(* CODESYS project EngineeringToolbox.library
   Company: Beckhoff Electronics Mfg
   DefaultNamespace: ET
   Version: 3.1.0.13
   Placeholder: ET
   Author: Daniel Schlingmann
   Description: Engineering Toolbox Library
      
      The library is provided "as-is" for TwinCAT3.1 by the Beckhoff Industry Management for Electronics Manufacturing.
      Please check the function "DisclaimerStatement : WSTRING[1500]"
   Title: EngineeringToolbox

Project tree, tasks and I/O mapping:
  libraries: Tc2_BackupRestoreEL6900, * (Beckhoff Automation GmbH); Tc2_Drive, * (Beckhoff Automation GmbH); Tc2_EtherCAT, * (Beckhoff Automation GmbH); Tc2_IoFunctions, * (Beckhoff Automation GmbH); Tc2_Math, * (Beckhoff Automation GmbH); Tc2_MC2, * (Beckhoff Automation GmbH); Tc2_MC2_Camming, * (Beckhoff Automation GmbH); Tc2_MC2_Drive, * (Beckhoff Automation GmbH); Tc2_MC2_FlyingSaw, * (Beckhoff Automation GmbH); Tc2_MDP, * (Beckhoff Automation GmbH); Tc2_ModbusRTU, * (Beckhoff Automation GmbH); Tc2_ModbusSrv, * (Beckhoff Automation GmbH); Tc2_NC, * (Beckhoff Automation GmbH); Tc2_NCI, * (Beckhoff Automation GmbH); Tc2_NcKinematicTransformation, * (Beckhoff Automation GmbH); Tc2_PlcInterpolation, * (Beckhoff Automation GmbH); Tc2_SerialCom, * (Beckhoff Automation GmbH); Tc2_Smtp, * (Beckhoff Automation GmbH); Tc2_Standard, * (Beckhoff Automation GmbH); Tc2_SUPS, * (Beckhoff Automation GmbH); Tc2_System, * (Beckhoff Automation GmbH); Tc2_TcpIp, * (Beckhoff Automation GmbH); Tc2_Utilities, * (Beckhoff Automation GmbH); Tc2_XmlDataSrv, * (Beckhoff Automation GmbH); Tc3_Module, * (Beckhoff Automation GmbH)
  GVLs/
    global variables Gvl
    global variables PARAM
  POUs/
    _Miscellaneous/
      64BitFunctions/
        function CLEARBIT64 [ST]
        function CSETBIT64 [ST]
        function GETBIT64 [ST]
        function SETBIT64 [ST]
      Conversions/
        function ADSERROR_TO_HRESULT [ST]
        function ADSERROR_TO_WIN32ERROR [ST]
        function ADSERROR_TO_WSERROR [ST]
        function C_TO_F [ST]
        function DEGREES_TO_RPM [ST]
        function DWORD_TO_REAL_EX [ST]
        function F_TO_C [ST]
        function GF_TO_N [ST]
        function HRESULT_TO_ADSERROR [ST]
        function LWORD_TO_LREAL_EX [ST]
        function MMIN_TO_MMS [ST]
        function MMS_TO_MMIN [ST]
        function N_TO_GF [ST]
        function REAL_TO_FMLREAL [ST]
        function RPM_TO_DEGREES [ST]
        function SWAP_BYTES_OF_WORDS [ST]
        function SWAP_WORDS_OF_DWORD [ST]
        function SWAP_WORDS_OF_LWORD [ST]
        function TO_FMLREAL [ST]
      function CAM [ST]
      function CAM3D [ST]
      data type COLOR
      data type eLCID
      function block ERROR_HDL [ST]: reset
      function block FbBase [ST]
      function block FbBaseExt [ST]
      function block FbBaseOutputs [ST]
      function getNoOfBits [ST]
      data type LCID
      function LOGx [ST]
      function nextIdx [ST]
      function block OEECalculation [ST]: addBadUnits, addGoodUnits, reset
      function polynomial [ST]
      function block RF_TRIG [ST]
      function scale [ST]
      function block SEQUENCE_HDL [ST]: abort, active, finish, incState, reset, resetWithErrHdl, set, ton_BT, ton_PT, tonOFF, tonON, tonRUN
      function setNoOfBits [ST]
      data type TC_VN_COLORS
      function block TEST_FB [ST]
      function block TOGGLE [ST]: CLK, RESET, SET
      data type U_32BIT_DATATYPE
      data type U_64BIT_DATATYPE
      function WIN [ST]
    BoundsCheck/
      function boundsError [ST]
      function boundsOK [ST]
      function block CheckBoundsInfo [ST]: reset, setErrorLower, setErrorUpper
    Connectivity/
      ADS/
        function block AdsDataExchange [ST]
      TF625x-Modbus/
        Master/
          _Components/
            function block ModbusJob [ST]: init
            function block ModbusSlaveCom [ST]: deleteData
          TF6250-ModbusTcpServer/
            TCP/
              function block ModbusTcpMaster [ST]: getNextJob, getNextSlave, reset, startJob
            UDP/
              function block ModbusUdpMaster [ST]: getNextJob, getNextSlave, reset, startJob
          TF6255-ModbusRtu/
            function block ModbusRtuMaster22B [ST]: getNextJob, getNextSlave, reset, startJob
            function block ModbusRtuMaster5B [ST]: getNextJob, getNextSlave, reset, startJob
            function block ModbusRtuMasterPC [ST]: getNextJob, getNextSlave, reset, startJob
        Slave/
          function block ModbusSlaveBase [ST]: evaluation, initJobs, prepareWriteData, run
      TF6310-TcpServer/
        TCP/
          function block TCPSendRecCtrl [ST]: optDoNotRestartReceiveCyclic, receive, send
          function block TCPServerCtrl [ST]
          function block TCPSocketCtrl [ST]: accept, close, closeAll, connect, listen
        UDP/
          function block UDPSendRecCtrl [ST]: optDoNotRestartReceiveCylic, receive, send
          function block UDPServerCtrl [ST]
          function block UDPSocketCtrl [ST]: close, closeAll, create
      TF6340-SerialCom/
        function block ComPortBackground [ST]: reset
        function block ComPortSendRec [ST]: clearBuffer, optClearBuffer, optEnableStringMode, optRemovePrefix, optRemoveSuffix, receiveData, receiveStr, reset, sendData, sendStr
      function isValidIPv4Addr [ST]
      data type U_IPv4Addr
    ControllerTools/
      function block AverageFilter [ST]: clear, insert
      function block PIDController [ST]: reset, synchronize
      function block PT1Filter [ST]: reset, synchronize
      function signum [ST]
      function block SlewRateLimitter [ST]: synchronize
      function block SlidingAverage [ST]: reset
      function block SlidingAverageExt [ST]: FB_exit, reset
      function block ThreePointController [ST]: reset, synchronize
    DataBuffer/
      Fifo/
        function block Fifo [ST]: clear, clearByDataSet, dequeue, enqueue, isEnqueued, isNextEntry, readEntry, reset
        function block FifoBase [ST]: _clear, _clearByDataSet, _dequeue, _enqueue, _isEnqueued, _isNextEntry, _readEntry, _reset
        function block FifoExt [ST]: allocate, clear, clearByDataSet, dequeue, enqueue, FB_exit, isEnqueued, isNextEntry, readEntry, reset
        function block FifoLRealSimple [ST]: clear, clearByDataSet, dequeue, enqueue, isEnqueued, isNextEntry, readEntry, reset
      Ringbuffer/
        function block Ringbuffer [ST]: dequeue, dequeueStream, enqueue, enqueueStream, reset
        function block RingbufferBase [ST]: _dequeue, _dequeueStream, _enqueue, _enqueueStream, _reset
        function block RingbufferByteSimple [ST]: dequeue, dequeueStream, enqueue, enqueueStream, reset
        function block RingbufferCharSimple [ST]: dequeue, dequeueStream, enqueue, enqueueStream, reset
        function block RingbufferExt [ST]: allocate, dequeue, dequeueStream, enqueue, enqueueStream, FB_exit, reset
        function block RingbufferLRealSimple [ST]: dequeue, dequeueStream, enqueue, enqueueStream, reset
      function block DataFileLogger [ST]: addData, addString, optKeepFileOnError, optStartNewFile
      function block DoubleBuffer [ST]: addData, addString, allocate, copyData, FB_exit, fillLevel, reset, setReadyToRead, swapBuffer
      function block Quicksort [ST]: allocate, byDINT, byDINT_Bubble, byINT, byLREAL, byLTIME, byREAL, bySTRING, byTIME, byUINT, byUSINT, byWSTRING, FB_exit
    EventLogger/
      ReadEvents/
        data type EVENTLOG_READ_DATA
        data type EVENTLOG_READ_HANDLEINFO
        data type EVENTLOG_READ_STREAM
        data type EVENTLOG_READ_STREAM_DATA_RAW
        data type EVENTLOG_READ_STREAM_DATA_RAW_EX
        function block EventlogRead [ST]: optGetHostNameForEachEvent, optUseStateForTimestamp
      TriggerEvents/
        function block EventHandling [ST]
        function EventHandlingConfirmIsReq [ST]
        function block EventHandlingGrp10 [ST]: confirm, confirmIsReq, isActive
        function block EventHandlingGrp25 [ST]: confirm, confirmIsReq, isActive
        function block EventHandlingGrp50 [ST]: confirm, confirmIsReq, isActive
        function block EventHandlingGrpCustomized [ST]: confirm
        function block EventHandlingStatisticInfo [ST]: classAlarmActive, classHintActive, classInstructionActive, classMaintenanceActive, classMessageActive, classNoneActive, classParamErrorActive, classStateinfoActive, classWarningActive, clear, countIn, countOut, initEvent, isClassActive, isConfirmReqActive, isPriorityActive
      data type EVENT_HANDLING_CONFIG
      function block EventsWriteToLogbook [ST]: _formatMsg
      function getEventClassPriority [ST]
      function getEventClassText [ST]
      data type SOURCE_ID
    Fieldbus/
      CANopen/
        function block CANopenMasterDiag [ST]
        function block CANopenMasterIO [ST]: setName
      EtherCAT/
        _Components/
          data type EC_MASTER_DEVICE_STATE
          data type EC_SLAVE_DIAG_INFO_DATA
          function block EcMasterIO [ST]
          function block EcMasterSupervisor [ST]: optClearCRCErrorCounter, optClearLostFramesCounter, optClearTCRXErrCounter, optForceDevReset
          function block EcSlavesDiag [ST]: allocate, FB_exit, optReadScannedSlaves, optSortInfoData, optUpdateConfigData, optUpdateTopoData, sortList
          function block EcSlaveSupervisor [ST]
        function block EcCoEReadNewestDiagMsg [ST]: msgSevyIsError, msgSevyIsInfo, msgSevyIsWarning
        function block EcDiagBase [ST]
        function block EcDiagBase_wEvents [ST]: _callEvents, confirm
      Profibus/
        function block ProfibusMasterDiag [ST]
        function block ProfibusMasterIO [ST]
      Profinet/
        function block ProfinetControllerIO [ST]
        function block ProfinetControllerIO_wEvents [ST]
        function block ProfinetDeviceIO [ST]
    FileHandling/
      Basic/
        function block FileHandling [ST]: close, createDir, delete, gets, isEoF, open, puts, read, removeDir, rename, seek, tell, write
        function block ReadDirSimple [ST]
        function block ReadDirSimpleExt [ST]
      TF6421-XmlServer/
        function block XmlReadWrite [ST]: read, write
        function block XmlReadWriteWithBackupFile [ST]: FB_exit, optEnableAutoSave, optEnableBackupFile, read, write
    IO/
      _EcSlaveFWUpdater/
        function block EcSlaveDevFWUpdater [ST]
      _EcSlaveInfoDataIO/
        function block EcSlaveInfoData [ST]: rInfoData
        function block EcSlaveInfoDataExt [ST]
        interface I_EcSlaveInfoData: rInfoData
      _ItfActuators/
        interface I_ActuatorBase: inError, isBusy, isOff, noFeed, ok, reset, switchOff
        interface I_ActuatorEnableDisable: isDisabled, isEnabled, setDisable, setEnable
        interface I_ActuatorFwdBwd: backwardStarted, forwardStarted, startBackward, startForward
        interface I_ActuatorFwdRev: forwardStarted, reverseStarted, startForward, startReverse
        interface I_ActuatorLeftRight: leftOk, rightOk, toTheLeft, toTheRight
        interface I_ActuatorOnOff: isOn, switchOn
        interface I_ActuatorOpenClose: isClosed, isOpened, setClose, setOpen
        interface I_ActuatorPosNeg: negativeOk, negativeOn, positiveOk, positiveOn
        interface I_ActuatorStartStop: isStarted, isStopped, start, stop
        interface I_ActuatorUpDown: downOk, moveDown, moveUp, upOK
        interface I_ActuatorWorkBase: isInBasePos, isInWorkPos, moveToBasePos, moveToWorkPos
      Cylinder/
        function block Cylinder [ST]: _readSensors, _runtimeChk, _writeStatus, enable, moveToBasePos, moveToWorkPos, reset, switchOff, optDisableLogicError, optDisableSensorBasepos, optDisableSensorWorkpos, optEnableImpulsValveFnc, optInvertSensorBasepos, optInvertSensorWorkpos, optSwapSensorStatus, inError, isBusy, isInBasePos, isInWorkPos, isOff, noFeed, ok, rCylinder, simulation
        function block CylinderExt [ST]: _runtimeChk
        function block CylinderType4 [ST]: _readSensors
        interface I_Cylinder: enable, rCylinder, simulation
      Drives/
        CoE/
          EL72xx/
            function block AxDriveCoE [ST]
            function block AxDriveCoE_EL72xxParam [ST]: deviceAddrIsValid, getValue, seqRead, seqWrite, setValue
            function block AxDriveCoE_wEvents [ST]: _callEvents, confirm, optDisabledRemoteCntrNotActive, optDisableIntLimitWarning
            function block CiA_DS402StatuswordEx7xxx [ST]: readStatusword
          function block CiA_DS402Controlword [ST]: createControlword
          function block CiA_DS402Statusword [ST]: readStatusword
          data type eCiA_DS402_CONTROL_CMD
          data type eCiA_DS402_STATUS_STATE
        DC/
          Ey73xx/
            function block AxDriveDC [ST]
            function block AxDriveDC_wEvents [ST]: _callEvents, confirm
        SoE/
          Ax5000ParamSTRUCTs/
            P/
              data type AX5000_P_0001
              data type AX5000_P_0002
              data type AX5000_P_0003
              data type AX5000_P_0004
              data type AX5000_P_0009
              data type AX5000_P_0010
              data type AX5000_P_0020
              data type AX5000_P_0021
              data type AX5000_P_0040
              data type AX5000_P_0050
              data type AX5000_P_0051
              data type AX5000_P_0052
              data type AX5000_P_0053
              data type AX5000_P_0054
              data type AX5000_P_0055
              data type AX5000_P_0056
              data type AX5000_P_0057
              data type AX5000_P_0058
              data type AX5000_P_0059
              data type AX5000_P_0060
              data type AX5000_P_0061
              data type AX5000_P_0062
              data type AX5000_P_0063
              data type AX5000_P_0064
              data type AX5000_P_0065
              data type AX5000_P_0066
              data type AX5000_P_0067
              data type AX5000_P_0068
              data type AX5000_P_0069
              data type AX5000_P_0070
              data type AX5000_P_0071
              data type AX5000_P_0072
              data type AX5000_P_0073
              data type AX5000_P_0074
              data type AX5000_P_0075
              data type AX5000_P_0076
              data type AX5000_P_0077
              data type AX5000_P_0078
              data type AX5000_P_0088
              data type AX5000_P_0089
              data type AX5000_P_0090
              data type AX5000_P_0091
              data type AX5000_P_0092
              data type AX5000_P_0093
              data type AX5000_P_0096
              data type AX5000_P_0097
              data type AX5000_P_0098_beckhoff
              data type AX5000_P_0098_beckhoff_electrical_data
              data type AX5000_P_0099
              data type AX5000_P_0100
              data type AX5000_P_0101
              data type AX5000_P_0102
              data type AX5000_P_0103
              data type AX5000_P_0104
              data type AX5000_P_0105
              data type AX5000_P_0106
              data type AX5000_P_0107
              data type AX5000_P_0108
              data type AX5000_P_0109
              data type AX5000_P_0110
              data type AX5000_P_0111
              data type AX5000_P_0112
              data type AX5000_P_0113
              data type AX5000_P_0114
              data type AX5000_P_0115
              data type AX5000_P_0116
              data type AX5000_P_0117
              data type AX5000_P_0118
              data type AX5000_P_0119
              data type AX5000_P_0125
              data type AX5000_P_0126
              data type AX5000_P_0127
              data type AX5000_P_0128
              data type AX5000_P_0150
              data type AX5000_P_0151
              data type AX5000_P_0152
              data type AX5000_P_0153
              data type AX5000_P_0154
              data type AX5000_P_0155
              data type AX5000_P_0158
              data type AX5000_P_0159
              data type AX5000_P_0160
              data type AX5000_P_0161
              data type AX5000_P_0162
              data type AX5000_P_0163
              data type AX5000_P_0165
              data type AX5000_P_0166
              data type AX5000_P_0167
              data type AX5000_P_0168
              data type AX5000_P_0169
              data type AX5000_P_0170
              data type AX5000_P_0171
              data type AX5000_P_0180
              data type AX5000_P_0181
              data type AX5000_P_0182
              data type AX5000_P_0183
              data type AX5000_P_0184
              data type AX5000_P_0185
              data type AX5000_P_0188
              data type AX5000_P_0189
              data type AX5000_P_0192
              data type AX5000_P_0193
              data type AX5000_P_0196
              data type AX5000_P_0198
              data type AX5000_P_0199
              data type AX5000_P_0200
              data type AX5000_P_0201
              data type AX5000_P_0202
              data type AX5000_P_0203
              data type AX5000_P_0204
              data type AX5000_P_0205
              data type AX5000_P_0206
              data type AX5000_P_0207
              data type AX5000_P_0208
              data type AX5000_P_0209
              data type AX5000_P_0210
              data type AX5000_P_0211
              data type AX5000_P_0212
              data type AX5000_P_0213
              data type AX5000_P_0214
              data type AX5000_P_0215
              data type AX5000_P_0216
              data type AX5000_P_0217
              data type AX5000_P_0218
              data type AX5000_P_0219
              data type AX5000_P_0220
              data type AX5000_P_0221
              data type AX5000_P_0250
              data type AX5000_P_0251
              data type AX5000_P_0252
              data type AX5000_P_0253
              data type AX5000_P_0254
              data type AX5000_P_0255
              data type AX5000_P_0256
              data type AX5000_P_0270
              data type AX5000_P_0271
              data type AX5000_P_0272
              data type AX5000_P_0273
              data type AX5000_P_0274
              data type AX5000_P_0275
              data type AX5000_P_0276
              data type AX5000_P_0277
              data type AX5000_P_0278
              data type AX5000_P_0300
              data type AX5000_P_0301
              data type AX5000_P_0302
              data type AX5000_P_0303
              data type AX5000_P_0304
              data type AX5000_P_0305
              data type AX5000_P_0306
              data type AX5000_P_0307
              data type AX5000_P_0308
              data type AX5000_P_0309
              data type AX5000_P_0310
              data type AX5000_P_0311
              data type AX5000_P_0312
              data type AX5000_P_0313
              data type AX5000_P_0314
              data type AX5000_P_0315
              data type AX5000_P_0316
              data type AX5000_P_0317
              data type AX5000_P_0320
              data type AX5000_P_0321
              data type AX5000_P_0322
              data type AX5000_P_0323
              data type AX5000_P_0324
              data type AX5000_P_0325
              data type AX5000_P_0326
              data type AX5000_P_0350
              data type AX5000_P_0351
              data type AX5000_P_0352
              data type AX5000_P_0353
              data type AX5000_P_0354
              data type AX5000_P_0356
              data type AX5000_P_0360
              data type AX5000_P_0361
              data type AX5000_P_0400
              data type AX5000_P_0401
              data type AX5000_P_0402
              data type AX5000_P_0451
              data type AX5000_P_0452
              data type AX5000_P_0453
              data type AX5000_P_0454
              data type AX5000_P_0455
              data type AX5000_P_0456
              data type AX5000_P_0457
              data type AX5000_P_0458
              data type AX5000_P_0459
              data type AX5000_P_0460
              data type AX5000_P_0461
              data type AX5000_P_0462
              data type AX5000_P_0463
              data type AX5000_P_0464
              data type AX5000_P_0502
              data type AX5000_P_0503
              data type AX5000_P_0504
              data type AX5000_P_0505
              data type AX5000_P_0511
              data type AX5000_P_0512
              data type AX5000_P_0513
              data type AX5000_P_0514
              data type AX5000_P_0515
              data type AX5000_P_0516
              data type AX5000_P_0517
              data type AX5000_P_0518
              data type AX5000_P_0552
              data type AX5000_P_0553
              data type AX5000_P_0554
              data type AX5000_P_0555
              data type AX5000_P_0556
              data type AX5000_P_0557
              data type AX5000_P_0558
              data type AX5000_P_0601
              data type AX5000_P_0602
              data type AX5000_P_0610
              data type AX5000_P_0611
              data type AX5000_P_0800
              data type AX5000_P_0801
              data type AX5000_P_0802
              data type AX5000_P_0804
              data type AX5000_P_0805
              data type AX5000_P_0806
              data type AX5000_P_0810
              data type AX5000_P_0811
              data type AX5000_P_0850
              data type AX5000_P_0851
              data type AX5000_P_0900
              data type AX5000_P_0901
              data type AX5000_P_0902
              data type AX5000_P_0904
              data type AX5000_P_0905
              data type AX5000_P_0906
              data type AX5000_P_0912
              data type AX5000_P_1000
              data type AX5000_P_1001
              data type AX5000_P_1002
              data type AX5000_P_1003
              data type AX5000_P_1004
              data type AX5000_P_1005
              data type AX5000_P_1006
              data type AX5000_P_1007
              data type AX5000_P_1008
              data type AX5000_P_1009
              data type AX5000_P_1010
              data type AX5000_P_1011
              data type AX5000_P_1012
              data type AX5000_P_1020
              data type AX5000_P_1021
              data type AX5000_P_1022
              data type AX5000_P_2000
              data type AX5000_P_2001
              data type AX5000_P_2002
            S/
              data type AX5000_S_0001
              data type AX5000_S_0002
              data type AX5000_S_0007
              data type AX5000_S_0011
              data type AX5000_S_0012
              data type AX5000_S_0013
              data type AX5000_S_0015
              data type AX5000_S_0016
              data type AX5000_S_0017
              data type AX5000_S_0018
              data type AX5000_S_0024
              data type AX5000_S_0029
              data type AX5000_S_0030
              data type AX5000_S_0031
              data type AX5000_S_0032
              data type AX5000_S_0033
              data type AX5000_S_0034
              data type AX5000_S_0035
              data type AX5000_S_0036
              data type AX5000_S_0037
              data type AX5000_S_0040
              data type AX5000_S_0043
              data type AX5000_S_0044
              data type AX5000_S_0045
              data type AX5000_S_0046
              data type AX5000_S_0047
              data type AX5000_S_0048
              data type AX5000_S_0051
              data type AX5000_S_0053
              data type AX5000_S_0055
              data type AX5000_S_0076
              data type AX5000_S_0079
              data type AX5000_S_0080
              data type AX5000_S_0081
              data type AX5000_S_0082
              data type AX5000_S_0083
              data type AX5000_S_0084
              data type AX5000_S_0085
              data type AX5000_S_0086
              data type AX5000_S_0091
              data type AX5000_S_0092
              data type AX5000_S_0095
              data type AX5000_S_0099
              data type AX5000_S_0100
              data type AX5000_S_0101
              data type AX5000_S_0103
              data type AX5000_S_0104
              data type AX5000_S_0106
              data type AX5000_S_0107
              data type AX5000_S_0109
              data type AX5000_S_0110
              data type AX5000_S_0111
              data type AX5000_S_0112
              data type AX5000_S_0113
              data type AX5000_S_0119
              data type AX5000_S_0120
              data type AX5000_S_0124
              data type AX5000_S_0126
              data type AX5000_S_0130
              data type AX5000_S_0131
              data type AX5000_S_0134
              data type AX5000_S_0135
              data type AX5000_S_0136
              data type AX5000_S_0137
              data type AX5000_S_0143
              data type AX5000_S_0149
              data type AX5000_S_0159
              data type AX5000_S_0160
              data type AX5000_S_0161
              data type AX5000_S_0162
              data type AX5000_S_0163
              data type AX5000_S_0169
              data type AX5000_S_0170
              data type AX5000_S_0179
              data type AX5000_S_0185
              data type AX5000_S_0186
              data type AX5000_S_0187
              data type AX5000_S_0188
              data type AX5000_S_0189
              data type AX5000_S_0196
              data type AX5000_S_0200
              data type AX5000_S_0201
              data type AX5000_S_0203
              data type AX5000_S_0204
              data type AX5000_S_0206
              data type AX5000_S_0207
              data type AX5000_S_0216
              data type AX5000_S_0217
              data type AX5000_S_0219
              data type AX5000_S_0254
              data type AX5000_S_0256
              data type AX5000_S_0257
              data type AX5000_S_0267
              data type AX5000_S_0273
              data type AX5000_S_0274
              data type AX5000_S_0292
              data type AX5000_S_0295
              data type AX5000_S_0296
              data type AX5000_S_0347
              data type AX5000_S_0348
              data type AX5000_S_0372
              data type AX5000_S_0374
              data type AX5000_S_0375
              data type AX5000_S_0380
              data type AX5000_S_0381
              data type AX5000_S_0383
              data type AX5000_S_0384
              data type AX5000_S_0390
              data type AX5000_S_0403
              data type AX5000_S_0405
              data type AX5000_S_0409
              data type AX5000_S_0410
              data type AX5000_S_0429
              data type AX5000_S_0432
              data type AX5000_S_0435
              data type AX5000_S_0436
          function block Ax580x [ST]
          function block AxDriveSoE_Ax5000 [ST]: break, refreshStatus, reset
          function block AxDriveSoE_Ax5000CalcPower [ST]: get_P_WORD, get_S_WORD
          function block AxDriveSoE_Ax5000CommutationCalib [ST]: optP98IsEmpty, optReadOnly
          function block AxDriveSoE_Ax5000Param [ST]: deviceAddrIsValid, getValue, seqRead, seqWrite, setValue
          function block AxDriveSoE_Ax5000SwitchParamSet [ST]: setNewParam
          function block AxDriveSoE_Ax5000wEvents [ST]: _callEvents, confirm
          function block AxDriveSoE_Rexroth [ST]: refreshStatus, reset, writeReferenz
        Stepper/
          function block AxDriveStepper [ST]
          function block AxDriveStepper_wEvents [ST]: _callEvents, confirm
          function block AxDriveStepperParam [ST]: deviceAddrIsValid, getValue, seqRead, seqWrite, setValue
        function block AxDriveBase [ST]: rAxDrive, rInfoData
        function block AxDriveGetRef [ST]
        interface I_AxDriveBase: rAxDrive
      EL-EP/
        EL3403/
          function block EL3403 [ST]
          function block EL3403Logic [ST]: readVariantValues
        EL9x/
          function block EL95xxPowerTerminal [ST]
          function block ELSystemTerminal [ST]
        EP92xxPwrBox/
          function block EP9214 [ST]: channelErrorUp, channelErrorUs, channelWarningUp, channelWarningUs
          function block EP9214_CHANNEL [ST]
          function block EP9224_0037 [ST]: channelErrorUp, channelErrorUs, channelWarningUp, channelWarningUs
          function block EP9224_0037_CHANNEL [ST]
        function block AnalogOut_EL2535 [ST]
        function block EL1904 [ST]
        function block EL3356 [ST]: inError, Q, Q_GramToNewton, Q_NewtonToGram
        function block EL69xx [ST]
        function block EL9576 [ST]
        function block Eyx9xx [ST]: inStateCrcOK, inStateError, inStateOffline, inStatePrepare, inStateRestore, inStateRun, inStateSafe, inStateStart, inStateStop
        function block ZB8610 [ST]: mode1Hz, mode2Hz, mode3Hz, mode4Hz, mode5Hz, mode6Hz, mode7Hz, mode8Hz, mode9Hz, modeHigh, modeTemp
      FreqConv/
        EtherCAT/
          DS402/
            function block EcFcDS402_ComBase [ST]: reset, setContactorOFF, setContactorON, setDisable, setEnable, switchOff, switchOn, inError, isBusy, isDisabled, isEnabled, isOff, isOn, noFeed, ok
        function block IOFcCom [ST]: closeBreak, openBreak, reset, setContactorOFF, setContactorON, startForward, startReverse, switchOff, switchOn, forwardStarted, inError, isBusy, isOff, isOn, noFeed, ok, reverseStarted
      Motors/
        function block IOMotor [ST]: _writeStatus, enable, reset, switchOff, switchOn, inError, isBusy, isOff, isOn, noFeed, ok
        function block IOMotor2Dir [ST]: _writeStatus, startForward, startReverse, switchOff, switchOn, forwardStarted, isOff, isOn, noFeed, reverseStarted
        function block IOMotorStarDelta [ST]: _writeStatus, reset, resetRestartTmr, switchOff, switchOn, isOn, ok
      function block AnalogIn [ST]: optEnableScaleSignedValue
      function block AnalogIn32 [ST]: optEnable24BitResolution, optEnableScaleExtRangeMode, optEnableScaleSignedValue, optShiftValueBy8Bits
      function block AnalogInELMBase [ST]
      function block AnalogInELMSingleSampleDINT [ST]: FB_init, optEnableScaleExtRangeMode
      function block AnalogInELMSingleSampleREAL [ST]: FB_init, optEnableScaleExtRangeMode
      function block AnalogOut [ST]: optEnableScaleSignedValue
      function block BlowOffSensors [ST]
      function block Button [ST]: setDisable, setEnable, setLedOFF, setLedON, TGL, TglOff, TglOn
      function block ButtonExt [ST]
      function block Fuse [ST]: reset
      function block InOut [ST]
      function block InOutExt [ST]: _runtimeChk, _writeStatus, enable, inError, isBusy, isOff, isOn, noFeed, ok, reset, switchOff, switchOn
      function block Input [ST]
      function block Output [ST]: switchOff, switchOn
    IpcDiag/
      MDP/
        InfoModuls/
          function block MDP_CPU [ST]
          function block MDP_Fan [ST]
          function block MDP_Mainboard [ST]
          function block MDP_RaidSimple [ST]
          function block MDP_ReadModulList [ST]
          function block MDP_SiliconDrives [ST]
          function block MDP_UPS [ST]
        function block MDP_Info [ST]: readAll, readCPU, readFan, readMB, readModList, readRaid, readSD, readUPS
        function block MDP_IpcDiag [ST]
        function block MDP_IpcDiag_wEvents [ST]: _callEvents
      function block UPSStatus [ST]
    Logging/
      function adsLogError [ST]
      function adsLogHint [ST]
      function adsLogWarn [ST]
      function adsLogwTcEventClass [ST]
      interface I_Logbook: delete, getOldestMsg, rCntAddedMessages, readMsg, write
      interface I_LogbookSubscriber: addNewMessage, isBusy
      function block Logbook [ST]: _write, delete, getOldestMsg, optAddDateToMsgText, optAddTimeToMsgText, optWiteEntryToTcAdsLogger, rCntAddedMessages, readMsg, write
      function block Logbook_wEventClass [ST]: getClassFromOption, write, writeWithClass
      data type LogbookData
      function block LogbookPuplisher [ST]: subscriberBusy
      function block LogbookSubEventLog [ST]: addNewMessage, FB_init, isBusy
      function block LogbookSubSendMail [ST]: addNewMessage, isBusy, optAddTimeToMsg, optEnableBufferError, optSendMsgIfDisabled
      function block LogbookSubSysLog [ST]: addNewMessage, createMsg, optAdd_CR, optAdd_LF, optEnabelDebugMode, optEnableBufferError, optEnableFacilitySeverityCode, optEnableRFCHeader, optSendMsgIfDisabled, isBusy
      function block LogbookSubWriteFile [ST]: addNewMessage, optAddDateToMsg, optAddEventClassToMsg, optAddTimeToMsg, optEnableBufferError, optSendMsgIfDisabled, optStartNewFile, isBusy
    Motion/
      TF50xx-NC/
        00_Base/
          function block AxFbBase [ST]
          function block AxRWParaBase [ST]: deviceAddrIsValid, read, seqRead, seqWrite, write
          interface I_AxNcBase: noAction, rAdmin, rAxisRef, rErrHdl, reset, rHome, rPara
          interface I_AxNcPTP: rMotion
        01_Main/
          function block AxAdmin [ST]: forceFeed, isResetting, isStopping, reset, seqEnable
          function block AxHoming [ST]: _MCIntern, cyclic, halt, homing, setPos
          function block AxMotion [ST]: _MCIntern, halt, jogOff, moveAbs, moveAdd, moveJog, moveMod, moveRel, moveVelo, stop
        02_Options/
          Coupling/
            function block AxCamming [ST]: camIn, camOut
            function block AxFlyingSaw [ST]: gearInPos, gearInVelo, gearOut
            function block AxGear [ST]: gearIn, gearInDyn, gearInMM, gearOut
          Error/
            function block AxEventHandling [ST]: confirm
            function block AxNcEventHandling [ST]
          Motion/
            function block AxHomingOnBlock [ST]
            function block AxMoveSinus [ST]
            function block AxSuperposition [ST]: moveAbort, moveImposed
          Parameter/
            function block AxPara [ST]: deviceAddrIsValid, getValue, seqRead, seqWrite, setValue
            function block AxParaCtrl [ST]: deviceAddrIsValid, getValue, seqRead, seqWrite, setValue
          Phasing/
            function block AxPhasing [ST]: haltPhasing, phasingAbsoulte, phasingRelative
          TouchProbe/
            function block AxTouchProbe [ST]: abort, run
        03_Utilities/
          function block AX_JOB [ST]: reset
          function block AxAutoFct [ST]
          function block AxAutoWriteSoftLimit [ST]
          function block AxCalcPosBias [ST]: optWritePosBiasToNC
          function block AxSoftSyncDistance [ST]
          function block AxStatemodel [ST]: aborted, aborting, clearing, completing, executing, resetting, starting, stateChanged, stopped, stopping
          function block CoordinateTransformation2D [ST]: diagonalMSC, diagonalPCS, isParamValid, MSCtoPCS, paramHasError, PCStoMSC
          function getOvrVelo [ST]
        function block AxNcBase [ST]: errorCheck, noAction, optEnableCmdAbortedAsError, rAdmin, rAxisRef, rErrHdl, reset, rHome, rPara
        function block AxNcBaseExt [ST]
        function block AxNcPTP [ST]: noAction, rMotion
        function block AxNcPtpGear [ST]: noAction, reset
        function block AxNcPTPwJobs [ST]: checkTargetPos, optEnableCyclicCheckTargetPos, startMotion
      TF5100-NCI/
        01_Main/
          function block NCI_REF [ST]: readStatus
          function block NciAdmin [ST]: reset, singleBlockModeChange, singleBlockTrigNext
          function block NciGrp [ST]: addAxis, build, reconfig, reconfigAxis
          function block NciItp [ST]: feedTbl, loadPrg, reset, startPrg, stopPrg
          function block NciMotion [ST]: disableFeederBackup, enableFeederBackup, eStop, retraceBwd, retraceFwd, stepOn
        02_Options/
          Error/
            function block NciChnEventHandling [ST]
            function block NciEventHandling [ST]: confirm
          MFunctions/
            function block NciMFnc [ST]: confirm, resetFastMFunc
          PlcItp/
            function block NciCreateItpTable [ST]: addCircleCIP, addDwellTime, addEndOfTable, addMFuncFast, addMFuncFastList, addMFuncHsk, addMFuncResetAllFast, reset, setAxisDynamics, setBaseFrame, setCirclePlane, setCoordinateSystem, setDynOverride, setGeoBezier3, setGeoBezier5, setGeoLine, setGeoStart, setHParam, setPathDynamics, setSParam, setTangFollowingDesc, setTParam, setVertexSmoothing
            function block NciCreateItpTableEntryTemplate [ST]: insertAxisDynamics, insertBaseFrame, insertDwellTime, insertDynOverride, insertEndOfTable, insertGeoBezier3, insertGeoBezier5, insertGeoCircleCIP, insertGeoCirclePlane, insertGeoLine, insertGeoStart, insertHParam, insertMFuncFast, insertMFuncHsk, insertMFuncResetAllFast, insertPathDynamics, insertSetCoordinateSystem, insertSParam, insertTangFollowingDesc, insertTParam, insertVertexSmoothing, reset
          RParameter/
            function block NCiReadWriteRParam [ST]: read, write
        function block NciChannel [ST]: noAction, reset
      TF511x-KIN/
        01_Main/
          function block KIN_REF [ST]: readStatus
          function block KinAdmin [ST]: reset
        02_Options/
          function block KinLockUnlockTrafoParam [ST]
          function block KinWriteToolTrafoParam [ST]
          function block KinWriteUCSTrafoParam [ST]
        03_DUTs/
          Positions/
            function block KIN_POSITIONS [ST]: copy, delete, isInPos, isInPosABC, isInPosByAxisNo, isInPosExt, isInPosXYZ, reset
            data type KIN_POSITIONS_ACS_DUT
            data type KIN_POSITIONS_MCS_DUT
            data type U_KIN_POSITIONS
          Trafo/
            function block KIN_CALCTRAFO_AXPOS_PARAM [ST]: delete
            function block KIN_STATE_OBSERVER_OID_PARAM [ST]: delete
            function block KIN_STATICTRAFO_PARAM [ST]: delete
            function block KIN_TOOLTRAFO_PARAM [ST]: delete
            function block UCS [ST]: delete
        function block KinChannel [ST]
      function block VALUE_3D [ST]: copy, delete, InPos, InPosByAxisNo, InPosXY, InPosXZ, InPosYZ, reset
      data type VALUE_3D_DUT
      function block VALUE_6D [ST]: copy, delete, inPos, InPosABC, InPosAC, inPosByAxisNo, inPosXY, InPosXYZ, inPosXZ, inPosYZ, reset
      data type VALUE_6D_DUT
    Safety/
      Diag/
        function block SafetyIODeviceDiag_wEvents [ST]: _eventsAX580x, _eventsConnDiag, _eventsDiagHistory, _eventsEK1914, _eventsEL2904, _eventsEx190x
        function block SafetyIODeviceDiagRead [ST]: FB_exit, msgSevyIsError, msgSevyIsInfo, msgSevyIsWarning
        function block SafetyIOsDiag [ST]
        function block SafetyLogicAndIOTerminalDiag [ST]: inputModuleFault, moduleInFault, outputModuleFault
        function block SafetyLogicTerminalDiag [ST]: FB_init, sourceId
        function block SafetyPlcTerminalDiag [ST]: FB_init
      data type SAFETY_CIRCUIT_STATUS
      function block SafetyCircuit [ST]
      function block SafetyGroupIO [ST]: diagCmpError, diagComError, diagDeactiveError, diagFbError, diagModuleError, diagNoError, diagRestartError, inStateDeactive, inStateError, inStateReset, inStateRun, inStateSafe, inStateStart, inStateStop, inStateStopError, inStateUnknow, inStateWaitComError
      function block SafetyPlcBackupRestore [ST]: backup, fileExists, restore
    Statemodel/
      control/
        interface I_Statemodel: addSlave, isModeActive, isStateActive, reset, setLocalError, remoteData, rErrHdl
        interface I_StatemodelBase: setMachineError, stateComplete, actMode, actState, isBusy, setStateComplete
        function block Statemodel [ST]: _createID, addSlave, FB_init, goToStopping, isModeActive, isStateActive, reset, setLocalError, setMachineError, stateComplete, optDisableSafetyInputs, optEnableAutoChangeModeToIdle, optEnableExplicitReset, optEnableExternalStateComplete, optEnableFwdMachineErrorToMaster, optEnableModeChangeInExecute, optEnableModeChangeViaStateCompl, optEnableSetActState, actMode, actState, ipMasterUnit, isBusy, remoteData, rErrHdl, setStateComplete
      UnitTemplate/
        interface I_Statemodel_Unit: rUnit
        function block Statemodel_Unit [ST]: aborted, aborting, clearing, complete, completing, executing, FB_exit, FB_init, FB_reinit, idle, resetting, rUnit, started, starting, startup, stateChanged, stopped, stopping
      data type eMODE
      data type eSTATE
    StringHelper/
      ExtendedString/
        function block ExtString [ST]: CONCAT, DELETE, FIND, INSERT, LEFT, LEN, MID, REPLACE, RIGHT
        function block ExtWString [ST]: CONCAT, DELETE, FIND, INSERT, LEFT, LEN, MID, REPLACE, RIGHT
        data type T_EXT_STRING
        data type T_EXT_WSTRING
      function cutStrNumberToSeperator [ST]
      function cutStrToSeperator [ST]
      function cutWStrToSeperator [ST]
      function DWORD_TO_BINSTR_EXT [ST]
      function DWORD_TO_HEXSTR_EXT [ST]
      function getCntCharInStr [ST]
      function getCntCharInWStr [ST]
      function getFilledString [ST]
      function HEXSTR_TO_DWORD [ST]
      function HEXSTR_TO_LWORD [ST]
      function INSERT_EXT [ST]
      function isStringNumeric [ST]
      function isWStringNumeric [ST]
      function LWORD_TO_BINSTR_EXT [ST]
      function LWORD_TO_HEXSTR_EXT [ST]
      function readStrToSeperator [ST]
      function readWStrToSeperator [ST]
      function replaceInString [ST]
      function replaceInWString [ST]
      function replaceUmlauts [ST]
      data type U_MAX_STRING
      data type U_MAX_WSTRING
      function WINSERT_EXT [ST]
    System/
      function block SystemInfo [ST]: actDCTimeWithTimezoneBias, optAddmsToTimeString, optDisableReadDeviceIdentification, optEnableUSDateFormat, optEnableUSTimeFormat, resetBootInfo, setSysTime
      function block SystemPulses [ST]: optAllOn, optEnable100ms, optEnable10m, optEnable10s, optEnable1m, optEnable1s, optEnable1s600msBlinkSlow, optEnable20ms, optEnable250msBlinkVeryFast, optEnable2s, optEnable400msBlinkFast, optEnable500ms, optEnable5m, optEnable5s, optEnable60m, optEnable800msBlink, optEnableCustom
      function block TaskInfo [ST]: resetCylceTimeExceeded
    TimeHelper/
      Conversions/
        function FILETIME_TO_DATE [ST]
        function FILETIME_TO_TOD [ST]
        function LREAL_TO_TIME_SEC [ST]
        function SYSTEMTIME_TO_DATE [ST]
        function SYSTEMTIME_TO_TIME [ST]
        function SYSTEMTIME_TO_TIME_EX [ST]
        function SYSTEMTIME_TO_TOD [ST]
        function TIME_TO_FMRLREAL [ST]
        function TIME_TO_SYSTEMTIME [ST]
      function createTOD [ST]
      function getDateAndTimeDelta [ST]
      function getTonCountdown [ST]
      function block LivebitCheck [ST]
      function block Ontime [ST]: reset
      function block OntimeExt [ST]: reset
      function block OntimeSimple [ST]: reset
      function block PartsPerTime [ST]: addNewPart, reset
      function block Pulse [ST]
      function block SensorTimeoutCheck [ST]: reset
      function block systemtimeCmp [ST]: dayOfWeek, days, hours, milliseconds, minutes, months, seconds, years
      function systemtimeInCam [ST]
      function systemtimeInWin [ST]
      function block TimeSwitch [ST]
      function block TONRecord [ST]: reset
      function block TONTOF [ST]: BT, reset
      function block VeloLinearMeasurement [ST]: reset
  Version/
    function disclaimerStatement [ST]
    global variables Global_Version
*)

// POUs/_Miscellaneous/COLOR
TYPE COLOR :
STRUCT
	NULL									: UDINT := 16#00000000;
	BLACK									: UDINT := 16#FF000000;	
	YELLOW									: UDINT := 16#FFFFFF00;
	RED										: UDINT := 16#FFFF0000;
	BLUE									: UDINT := 16#FF0000FF;
	GREEN									: UDINT := 16#FF008000;
	GREY									: UDINT := 16#FF808080;
	GREYDARK								: UDINT := 16#FFC0C0C0;
	PINK									: UDINT := 16#FFFFC0CB;
	ORANGE									: UDINT := 16#FFFFA500;
	VIOLET									: UDINT := 16#FFEE82EE;
	WHITE									: UDINT := 16#FFFFFFFF;																										
END_STRUCT
END_TYPE

// POUs/_Miscellaneous/eLCID
{attribute 'qualified_only'}
{attribute 'to_string'}
TYPE eLCID :
(
// Code: 	https://de.wikipedia.org/wiki/ISO-3166-1-Kodierliste
// LCID:	https://msdn.microsoft.com/de-de/goglobal/bb964664.aspx
// LCID:	https://winprotocoldoc.blob.core.windows.net/productionwindowsarchives/MS-LCID/%5bMS-LCID%5d.pdf

//	ISO3166 ALPHA-2
	NONE					:= 0,
	CZ						:= 1029, // Czech - 1029 
	DK						:= 1030, // Danish - 1030
	DE						:= 1031, // German - 1033
	GR						:= 1032, // Greek - 1032
	US						:= 1033, // English(US) - 1033
	ES						:= 1034, // Spanish(Spain) - 1034
	FI						:= 1035, // Finnish - 1035
	FR						:= 1036, // French(France) - 1036	
	IT						:= 1040, // Italian - 1040
	NL						:= 1043, // Dutch(Netherlands) - 1043
	NO						:= 1044, // Norwegian - 1044
	PL						:= 1045, // Polish - 1045
	RU						:= 1049, // Russian - 1049
	SE						:= 1053, // Swedish(Sweden) - 1053
	CA						:= 1099, // Canadian - 1099
	TR						:= 1055, // Turkish - 1055
	CN						:= 2052, // Chinese(CN-Simplified) - 2052
	GB						:= 2057, // English(UK) - 2057	
	PT						:= 2070 // Portuguese(Portugal) - 2057	
);
END_TYPE

// POUs/_Miscellaneous/LCID
{attribute 'qualified_only'}
TYPE LCID :
STRUCT
// Code: 	https://de.wikipedia.org/wiki/ISO-3166-1-Kodierliste
// LCID:	https://msdn.microsoft.com/de-de/goglobal/bb964664.aspx
// LCID:	https://winprotocoldoc.blob.core.windows.net/productionwindowsarchives/MS-LCID/%5bMS-LCID%5d.pdf

//	ISO3166 ALPHA-2, ALPHA-3
	NONE						: eLCID := eLCID.NONE;
	CZ,CZE						: eLCID := eLCID.CZ; // Czech - 1029 
	DK,DNK						: eLCID := eLCID.DK; // Danish - 1030
	DE,DEU						: eLCID := eLCID.DE; // German - 1033	
	GR,GRC						: eLCID := eLCID.GR; // Greek - 1032
	US,USA						: eLCID := eLCID.US; // English(US) - 1033
	ES,ESP						: eLCID := eLCID.ES; // Spainsh(Spain) - 1034
	FI,FIN						: eLCID := eLCID.FI; // Finnish - 1035
	FR,FRA						: eLCID := eLCID.FR; // French(France) - 1036	
	IT,ITA						: eLCID := eLCID.IT; // Italian - 1040
	NL,NLD						: eLCID := eLCID.NL; // Dutch(Netherlands) - 1043
	NO,NOR						: eLCID := eLCID.NO; // Norwegian - 1044
	PL,POL						: eLCID := eLCID.PL; // Polish - 1045
	RU,RUS						: eLCID := eLCID.RU; // Russian - 1049
	SE,SWE						: eLCID := eLCID.SE; // Swedish(Sweden) - 1053
	CA,CAN						: eLCID := eLCID.CA; // Canadian - 1099
	TR,TUR						: eLCID := eLCID.TR; // Turkish - 1055
	CN,CHN						: eLCID := eLCID.CN; // Chinese(CN-Simplified) - 2052
	GB,GBR						: eLCID := eLCID.GB; // English(UK) - 2057	
	PT,PRT						: eLCID := eLCID.PT; // Portuguese(Portugal) - 2057	
END_STRUCT
END_TYPE

// POUs/_Miscellaneous/TC_VN_COLORS
TYPE TC_VN_COLORS :
STRUCT
	// Colors
	BLACK		: TcVnVector4_LREAL := [0, 0, 0, 255];
	WHITE		: TcVnVector4_LREAL := [255, 255, 255, 255];
	RED			: TcVnVector4_LREAL := [255, 0, 0, 255];
	LIME		: TcVnVector4_LREAL := [0, 255, 0, 255]; //bright green
	BLUE		: TcVnVector4_LREAL := [0, 0, 255, 255];
	YELLOW		: TcVnVector4_LREAL := [255, 255, 0, 255];
	CYAN		: TcVnVector4_LREAL := [0, 255, 255, 255];	
	MAGENTA		: TcVnVector4_LREAL := [255, 0, 255, 255];
	SILVER		: TcVnVector4_LREAL := [192,192,192, 255];
	GRAY		: TcVnVector4_LREAL := [128,128,128, 255]; //darker than silver
	MAROON		: TcVnVector4_LREAL := [128,0,0, 255];
	OLIVE		: TcVnVector4_LREAL := [128,128,0, 255];
	GREEN		: TcVnVector4_LREAL := [0,128,0, 255]; //darker green
	PURPLE		: TcVnVector4_LREAL := [128,0,128, 255];
	TEAL		: TcVnVector4_LREAL := [0,128,128, 255];
	NAVY		: TcVnVector4_LREAL := [0,0,128, 255];
END_STRUCT
END_TYPE

// POUs/_Miscellaneous/U_32BIT_DATATYPE
TYPE U_32BIT_DATATYPE :  //Union datatype of 32 bit size datatypes 
UNION
	_REAL				: REAL;  
	{attribute 'displaymode':='hex'}	
	_DWORD				: DWORD;
	_DINT				: DINT;
	_UDINT				: UDINT;
	_TIME				: TIME;	
	_SINTS				: ARRAY[0..3] OF SINT; //Array 0..3 of BYTE
	{attribute 'displaymode':='hex'}	
	_BYTES				: ARRAY[0..3] OF BYTE; //Array 0..3 of BYTE
	{attribute 'displaymode':='hex'}	
	_WORDS				: ARRAY[0..1] OF WORD;	//Array 0..1 of WORD
	_INTS				: ARRAY[0..1] OF INT;	//Array 0..1 of INT
	_UINTS				: ARRAY[0..1] OF UINT;	//Array 0..1 of UINT
	
END_UNION
END_TYPE

// POUs/_Miscellaneous/U_64BIT_DATATYPE
TYPE U_64BIT_DATATYPE : //Union datatype of 64 bit size datatypes 
UNION
//Native 64bit data types
	_LREAL													:	LREAL; 
	_LINT													:	LINT;
	_ULINT													:	ULINT;
	_LTIME													:	LTIME;
	{attribute 'displaymode':='hex'}                         	
	_LWORD													:	LWORD;	
	                    
//Alternative 64bit size variables as arrays of smaller datatypes                                     	
	_DINTs				 									:	ARRAY[0..1] OF DINT; //Array 0..1 of DINT
	_UDINTs													:	ARRAY[0..1] OF UDINT; //Array 0..1 of UDINT
	_INTs													: 	ARRAY[0..3] OF INT;	//Array 0..3 of INT
	_UINTs													: 	ARRAY[0..3] OF UINT;//Array 0..3 of UINT 
	_SINTs													: 	ARRAY[0..7] OF SINT;//Array 0..7 of SINT (signed 8bit)
	{attribute 'displaymode':='hex'}	                     	
	_BYTEs													:	ARRAY[0..7] OF BYTE; //Array 0..7 of BYTE
	{attribute 'displaymode':='hex'}	                     	
	_WORDs													:	ARRAY[0..3] OF WORD; //Array 0..3 of WORD
	{attribute 'displaymode':='hex'}	                     	
	_DWORDs													:	ARRAY[0..1] OF DWORD; //Array 0..1 of DWORD
END_UNION
END_TYPE

// POUs/Connectivity/U_IPv4Addr
//IP v4 address as an union to provide the address in a UDINT and array format 
TYPE U_IPv4Addr : 
UNION
	Stacked 				: UDINT; //IPv4 address combined in a UDINT
	Bytes 					: T_IPv4AddrArr; //IPv4 address as an array 0..3 of Byte
END_UNION
END_TYPE

// POUs/EventLogger/ReadEvents/EVENTLOG_READ_DATA
TYPE EVENTLOG_READ_DATA :
STRUCT
	Class			: E_TcEventClass;	//See Beckhoff documentation for more information
	Computer		: STRING(80);		//Computer name of event source
	Timestamp		: T_DCTIME64;		//Timestamp in 64bit DC time format 
	TimestampDT		: DT;				//Timestamp in DATE_AND_TIME format 
	SourceId		: DWORD;			//Event Source ID
	id				: DWORD;			//Event number	
	State			: DWORD;			//Event state 
	Flags			: DWORD;			(*  TCEVENTFLAG_REQ=0x0001,
											TCEVENTFLAG_REQMUSTCON=0x0002,
											TCEVENTFLAG_CON=0x0004,
											TCEVENTFLAG_RESET=0x0008,
											TCEVENTFLAG_PRIOCLASS=0x0010,
											TCEVENTFLAG_FMTSELF=0x0020,
											TCEVENTFLAG_LOG=0x0040,
											TCEVENTFLAG_MSGBOX=0x0080,
											TCEVENTFLAG_SRCID=0x0100,
											TCEVENTFLAG_SELFRESET=0x0200,
											TCEVENTFLAG_TCID=0x0400,
											TCEVENTFLAG_SIGNAL=0x0800,
											TCEVENTFLAG_ADS=0x8000 *)
	Source			: WSTRING(40);		//Source name	
	MsgText			: WSTRING(255);		//Event message text in Unicode
	MegLen			: DWORD;			//Length of event message
END_STRUCT
END_TYPE

// POUs/EventLogger/ReadEvents/EVENTLOG_READ_HANDLEINFO
TYPE EVENTLOG_READ_HANDLEINFO :
STRUCT
	Enum			: DWORD;
	Count			: DWORD;
END_STRUCT
END_TYPE

// POUs/EventLogger/ReadEvents/EVENTLOG_READ_STREAM
TYPE EVENTLOG_READ_STREAM :
STRUCT
	cbStream		: DWORD; //size OF this structure, including all following TcGetEventParams structures
	count			: DWORD;
	data			: EVENTLOG_READ_STREAM_DATA_RAW;	(* Stream OF TcGetEventParams *)
END_STRUCT
END_TYPE

// POUs/EventLogger/ReadEvents/EVENTLOG_READ_STREAM_DATA_RAW
TYPE EVENTLOG_READ_STREAM_DATA_RAW :
STRUCT
	cb						: DWORD;	
	InvokeId				: DWORD;	
	Id						: DWORD;
	SrcId					: DWORD;
	AdsAddr					: ARRAY [0..5] OF BYTE;
	AddrHint				: ARRAY [0..1] OF BYTE;
	Class					: DWORD;
	Flags					: DWORD;
	Prio					: DWORD;
	State					: DWORD;
	UserData				: DWORD;
	zFmtProgId				: STRING(31);

	TimeSignaled			: T_FILETIME; //In UTC
	TimeReseted				: T_FILETIME; //In UTC
	TimeConfirmed			: T_FILETIME; //In UTC

	evtData					: EVENTLOG_READ_STREAM_DATA_RAW_EX;
	
END_STRUCT
END_TYPE

// POUs/EventLogger/ReadEvents/EVENTLOG_READ_STREAM_DATA_RAW_EX
TYPE EVENTLOG_READ_STREAM_DATA_RAW_EX :
STRUCT
	cb				: WORD;			//Complete size OF the structure including data
	cbFmt			: WORD;			//Size OF the format STRING
	cbData			: WORD;			//Size OF the data
	Temp			: ARRAY [PARAM.EVENT_HANDLING_CONFIG.EVENTLOG_READ_MSG_LEN_MIN..PARAM.EVENT_HANDLING_CONFIG.EVENTLOG_READ_MSG_LEN_MAX] OF BYTE;
	
END_STRUCT
END_TYPE

// POUs/EventLogger/EVENT_HANDLING_CONFIG
{attribute 'hide'}
//Library Param structure for EventLogger related function blocks  
TYPE EVENT_HANDLING_CONFIG :
STRUCT
	GRP_CUSTOMISED_MAX_EVENT								:	INT(1..1000) ;
	
	EVENTLOG_READ_MSG_LEN_MIN								:	INT(0..1) ;
	EVENTLOG_READ_MSG_LEN_MAX								:	INT(0..2096) ;	
                                                                     
	EVENTLOG_READ_MAX_EVENTS								:	INT(1..1000) ;
	                                                            
	ENABLE_DYNAMIC_EVENT_MSG_FORMAT							:	BOOL	; //Enable to adjust the placeholder (format) of the event messages according the use of Parameter EventHandling.Text1,Text2 and pText3
	
	CLASS_NONE_QUIT_REQUIRED								:	BOOL     ;
	CLASS_MAINTENANCE_QUIT_REQUIRED							:	BOOL     ;
	CLASS_MESSAGE_QUIT_REQUIRED								:	BOOL     ;
	CLASS_HINT_QUIT_REQUIRED								:	BOOL     ;
	CLASS_STATEINFO_QUIT_REQUIRED							:	BOOL     ;
	CLASS_INSTRUCTION_QUIT_REQUIRED							:	BOOL     ;
	CLASS_WARNING_QUIT_REQUIRED								:	BOOL     ;
	CLASS_ALARM_QUIT_REQUIRED								:	BOOL     ;
	CLASS_PARAMERROR_QUIT_REQUIRED							:	BOOL     ;
	                                                    	             
	CLASS_NONE_PRIORITY										:	UINT(0..3); //1=high ...3=low 
	CLASS_MAINTENANCE_PRIORITY								:	UINT(0..3); //1=high ...3=low 
	CLASS_MESSAGE_PRIORITY									:	UINT(0..3); //1=high ...3=low 
	CLASS_HINT_PRIORITY										:	UINT(0..3); //1=high ...3=low 
	CLASS_STATEINFO_PRIORITY								:	UINT(0..3); //1=high ...3=low 
	CLASS_INSTRUCTION_PRIORITY								:	UINT(0..3); //1=high ...3=low 
	CLASS_WARNING_PRIORITY									:	UINT(0..3); //1=high ...3=low 
	CLASS_ALARM_PRIORITY									:	UINT(0..3); //1=high ...3=low 
	CLASS_PARAMERROR_PRIORITY								:	UINT(0..3); //1=high ...3=low 
END_STRUCT
END_TYPE

// POUs/EventLogger/SOURCE_ID
{attribute 'qualified_only'}
//Predefined EventLogger Source Ids which collaborate to the default TcEventLogger Excel sheet   
//Most source IDs are already used as initial values for function blocks in this lib
TYPE SOURCE_ID :
STRUCT	
	TC_IO_MESSAGES			:	UDINT := 300;		//Reserved - TC3 default for TcIoMessages.xml
	TC_NC_MESSAGES			:	UDINT := 500;		//Reserved - TC3 default for TcNcMessages.xml
	TC_MIN_CNC_ERRORS		:	UDINT := 550;		//Reserved - TC3 default for TcCncErrors.xml
	TC_MAX_CNC_ERRORS		:	UDINT := 599;		//Reserved - TC3 default for TcCncErrors.xml
	TC_MIN_CNC_USER_EVENTS	:	UDINT := 650;		//Reserved - TC3 TcCncUserEvents.xml
	TC_MAX_CNC_USER_EVENTS	:	UDINT := 699;		//Reserved - TC3 TcCncUserEvents.xml
	TC_NC_DEF				:	UDINT := 700;		//Reserved - TC3 default for NCDefs.xml
	TC_NC_DEF_2				:	UDINT := 701;		//Reserved - TC3 default for NCDefs.xml
	
//	TcIoMessages.xml		:	UDINT := 300;		space - TC3 default 
//	TcNcMessages.xml		:	UDINT := 500;		space - TC3 default
//	TcCncErrors.xml			:	UDINT := 550-599;	space - TC3 default
//	TcCncUserEvents.xml		:	UDINT := 650-699;	space - TC3 default
//	NCDefs.xml				:	UDINT := 700-701;	space - NC Default
	
// 	General 0000- 0100
	GENERAL_STARTUP			:	UDINT := 100000;
	IPC_DIAG				:	UDINT := 100001;
	
// Safety 	0300-0399
	MIN_SAFETY_PLC_TERM_DIAG:	UDINT := 100300;
	MAX_SAFETY_PLC_TERM_DIAG:	UDINT := 100309;

	MIN_SAFETY_IO_TERM_DIAG	:	UDINT := 100310;
	MAX_SAFETY_IO_TERM_DIAG	:	UDINT := 100399;

// NC		1000-1999
	MIN_NC_AXIS				:	UDINT := 101000;	// NC Axis Min 
	MAX_NC_AXIS				:	UDINT := 101199;	// NC Axis Max
	
	MIN_NCI_GROUP			:	UDINT := 101200;	// NCI Groups Min 
	MAX_NCI_GROUP			:	UDINT := 101209;	// NCI Groups Max 
	
	MIN_KIN_GROUP			:	UDINT := 101210;	// Kinematik Groups Min 
	MAX_KIN_GROUP			:	UDINT := 101219;	// Kinematik Groups Max 
	
	MIN_XTS_GROUP			:	UDINT := 101220;	// XTS Groups Min 
	MAX_XTS_GROUP			:	UDINT := 101229;	// XTS Groups Max 
	
	MIN_CA_GROUP			:	UDINT := 101230;	// CA - Collision Avoidance Min 
	MAX_CA_GROUP			:	UDINT := 101239;	// CA - Collision Avoidance Max 
	
	MIN_PP_GROUP			:	UDINT := 101240;	// PP - Pick and Place Min 
	MAX_PP_GROUP			:	UDINT := 101249;	// PP - Pick and Place Max 

// Drives	2000-2999
	MIN_DRIVE_SOE			:	UDINT := 102000;	// Sercos Drive Min 
	MAX_DRIVE_SOE			:	UDINT := 102199;	// Sercos Drive Max 
	
	MIN_DRIVE_COE			:	UDINT := 102200;	// CanOpen Drive Min 
	MAX_DRIVE_COE			:	UDINT := 102399;	// CanOpen Drive Max 

	MIN_DRIVE_HYDR			:	UDINT := 102400;	// Hydraulic Drive Min 
	MAX_DRIVE_HYDR			:	UDINT := 102599;	// Hydraulic Drive Max 
	
	MIN_DRIVE_STEPPER		:	UDINT := 102600;	// Stepper Drive Min 
	MAX_DRIVE_STEPPER		:	UDINT := 102799;	// Stepper Drive Max 
	
// Fieldbus	3000-3099
	MIN_HW_EC_DIAG			:	UDINT := 103000;	// EtherCAT Master Min 
	MAX_HW_EC_DIAG			:	UDINT := 103009;	// EtherCAT Master Max 

	MIN_HW_CAN_DIAG			:	UDINT := 103010;	// CanOpen Master Min 
	MAX_HW_CAN_DIAG			:	UDINT := 103019;	// CanOpen Master Max 

	MIN_HW_PB_DIAG			:	UDINT := 103020;	// ProfiBus Master Min 
	MAX_HW_PB_DIAG			:	UDINT := 103029;	// ProfiBus Master Max 

	MIN_HW_PN_DIAG			:	UDINT := 103030;	// ProfiNet Master Min 
	MAX_HW_PN_DIAG			:	UDINT := 103039;	// ProfiNet Master Max 

	MIN_HW_DN_DIAG			:	UDINT := 103040;	// DeviceNet Master Min 
	MAX_HW_DN_DIAG			:	UDINT := 103049;	// DeviceNet Master Max 

	MIN_HW_S3_DIAG			:	UDINT := 103050;	// Sercos 3 Master Min 
	MAX_HW_S3_DIAG			:	UDINT := 103059;	// Sercos 3 Master Max 

	MIN_HW_LB_DIAG			:	UDINT := 103060;	// LightBus Master Min 
	MAX_HW_LB_DIAG			:	UDINT := 103069;	// LightBus Master Max 

	MIN_HW_IB_DIAG			:	UDINT := 103070;	// InterBus Master Min 
	MAX_HW_IB_DIAG			:	UDINT := 103079;	// InterBus Master Max 

	MIN_HW_EIP_DIAG			:	UDINT := 103080;	// Ethernet/IP Master Min 
	MAX_HW_EIP_DIAG			:	UDINT := 103089;	// Ethernet/IP Master Max 
	
END_STRUCT
END_TYPE

// POUs/Fieldbus/EtherCAT/_Components/EC_MASTER_DEVICE_STATE
TYPE EC_MASTER_DEVICE_STATE :
STRUCT
	NoError						: BOOL;//0x0000 = Link error 
	LinkError 					: BOOL;//0x0001 = Link error
	IOLockedAfterLinkError	    : BOOL;//0x0002 = I/O locked after link error (I/O reset required)
	LinkErrorRedMode			: BOOL;//0x0004 = Link error (redundancy adapter)
	MissingOneFrmInRedMode      : BOOL;//0x0008 = Missing one frame (redundancy mode)
	OutOfSendResources          : BOOL;//0x0010 = Out of send resources (I/O reset required)
	WatchdogTriggered 		    : BOOL;//0x0020 = Watchdog triggered
	EthernetDriverNotFound 	    : BOOL;//0x0040 = Ethernet driver (miniport) not found
	IOResetActive 			    : BOOL;//0x0080 = I/O reset active
	AtLeastOneSlaveInINIT       : BOOL;//0x0100 = At least one device in 'INIT' 
	AtLeastOneSlaveInPREOP      : BOOL;//0x0200 = At least one device in 'PRE-OP' 
	AtLeastOneSlaveInSAFEOP     : BOOL;//0x0400 = At least one device in 'SAFE-OP' 
	AtLeastOneSlaveInERROR     	: BOOL;//0x0800 = AT least one device indicates an error state 																	
	DcNotInSync 		        : BOOL;//0x1000 = DC NOT in sync
END_STRUCT
END_TYPE

// POUs/Fieldbus/EtherCAT/_Components/EC_SLAVE_DIAG_INFO_DATA
TYPE EC_SLAVE_DIAG_INFO_DATA :
STRUCT
	Addr									:	WORD; //Slaves own physical address e.g. 1004 
	ConfigType								:	STRING(18); //Configured type e.g. EL1008 or EL7211 
	ConfigName								:	STRING(31); //Name as configured in IO-tree (type removed)
	ConfigTypeIdentity						:	STRING(18); //Configured type according identity e.g. AX5206-0000-0210
	ScannedTypeIdentity						:	STRING(18); //Scanned type according identitiy e.g. EL7201-9014
	
//	{attribute 'displaymode':='hex'}  	
//	DevType									:	DWORD; //EtherCAT device type of a slave
	{attribute 'displaymode':='hex'}  
	DevState								:	BYTE; //Device state constant e.g. 16#08=Tc2_EtherCAT.EC_DEVICE_STATE_OP
	DevStateText							:	STRING(60); //e.g. OP, INIT etc...
	DevStateBits							:	ST_EcSlaveStateBitsEx; //The structure contains bits showing the EtherCAT status (e.g. OP) and the link status )e.g. (EC_LINK_STATE_MISSING_LINK)

	{attribute 'displaymode':='hex'}  
	LinkState								:	BYTE; //Link state constant e.g. 0=Tc2_EtherCAT.EC_LINK_STATE_NOT_PRESENT
	{attribute 'displaymode':='bin'}  
	DataLinkStatusReg						:	WORD; //Data link status register status based on Topology of an EtherCAT slave from ESC register 0110/0111hex or 272/273dec. Status 0 is displayed if the slave cannot be reached or is offline	

	//Error information	
	CntOfCRCErrors							:	UDINT; //Total number of CRC-Errors on all four ports of the slave 
	NoOfAbnormalStateChanges				:	UDINT; //Shows how many times the slave status changed from available to INIT_NO_COMM e.g. unpluged
	
	//Topology information
	HotConnectNodeStart						:	BOOL; //Indicates that slaves is teh start of a hot-connect group (bit.3 of topology status)
	HotConnectSlave							:	BOOL; //Indicates that the slave is a part of a hot-connect group (bit.4 of topology status)
   	HCSlaveCountCfg  						:  UINT; //Shows number of attached slaves at HC node start
 	HCSlaveCountAct  						:  UINT; //Shows number of active slaves at HC node start
	{attribute 'displaymode':='bin'}  
	TopologyStatus					      	:  DWORD; (* Bits.0 = TRUE: Distributed clocks are supported
														 Bits.1 = TRUE: Distributed clocks are supported (64 bit)
														 Bits.2 = TRUE: Slave is present
														 Bits.3 = TRUE: Slave is start node of a Hot Connect group
														 Bits.4 = TRUE: Slave is in a Hot Connect group
														 Bits.5 = TRUE: Hot-connect is invalid at port B
														 Bits.6 = TRUE: Hot-connect is invalid at port C
														 Bits.7 = TRUE: Hot-connect is invalid at port D *)

   	TopoOwnPhysicalAddr  					:  UINT; //Can be different to "Addr" automatically assigned
   	AutoIncAddr   							:  UINT; //Dedicated auto-increment address of slave
   	PhysicalPortAddr    					:  ST_PortAddr; //Structure with phy. addr. information at port A…D
   	AutoIncPortAddr    				 		:  ST_PortAddr; //Structure with Auto inc. addr. information at port A…D
	ConfigIdentity							:	ST_EcSlaveIdentity; //EtherCAT identity data of an EtherCAT slave device, vendor Id, product code etc...
	ScannedIdentity							:	ST_EcSlaveIdentity; //EtherCAT identity data of an EtherCAT slave device, vendor Id, product code etc...
	
	ScannedSeq								:	UINT; //Logical/scanned sequence which can be different to configured seq. if hot-connect groups are used 
	{attribute 'displaymode':='bin'}   
	ErrorIdentCode							:	WORD; //Interal error identefier (Not in OP, CRC error increased, etc...
END_STRUCT
END_TYPE

// POUs/IO/Drives/CoE/eCiA_DS402_CONTROL_CMD
{attribute 'qualified_only'}
{attribute 'to_string'}
TYPE eCiA_DS402_CONTROL_CMD :
(
	IDLE													:= 2#0000_0000, //2#0000_0000
	SHUTDOWN												:= 2#0000_0110, //2#0xxx_x110 -> Ready to switch on(Enable Voltage)
 	SWITCH_ON												:= 2#0000_0111, //2#0xxx_0111 -> Switched On (Switch on + Disable operation)
	DISABLE_VOLTAGE											:= 2#0000_0010, //2#0xxx_xx0x -> back to switch on disabled
	ENABLE_OPERATION										:= 2#0000_1111, //2#0xx0_1111 -> Operation enabled (Enable Voltage + Switch on + Enable operation)
	FAULT_RESET												:= 2#1000_0000, //2#1xxx_xxxx 
	QUICK_STOP												:= 2#1000_0010 //2#0xxx_x01x 
);
END_TYPE

// POUs/IO/Drives/CoE/eCiA_DS402_STATUS_STATE
{attribute 'qualified_only'}
{attribute 'to_string'}
TYPE eCiA_DS402_STATUS_STATE :
(
	NOT_READY_TO_SWITCH_ON									:= 2#0000_0000, //2#x0xx_0000 / Not ready to switch on. The drive is initialising or being configured.
	SWITCH_ON_DISABLED										:= 2#0100_0000, //2#x1xx_0000 / The Drive will not accept a switch on command 
	READY_TO_SWITCH_ON										:= 2#0010_0001, //2#x01x_0001 / The Drive will accept a switch on command.
	SWITCHED_ON												:= 2#0010_0011, (* 2#x01x_0011 / The Drive will accept an Operation Enable (Run or Jog) command. 		
																				- Power stage of the Drive is ready to operate.
																				- Voltage has not yet been applied to the motor terminals*)
	OPERATION_ENABLED										:= 2#0010_0111,  (* 2#x01x_0111 / Normal operational state of the drive. This state includes Running, Jogging,
																				Stopping (Disabling Operation) and Shutting Down (Switching Off).
																				- Voltage applied to the motor terminals. *)
	QUICK_STOP_ACTIVE										:= 2#0000_0111, //2#x00x_0111 / Emergency stop (Fast stop) is active
    FAULT_REACTION_ACTIVE									:= 2#0000_1111, //2#x0xx_1111 / The Drive is processing a tripped event                                                                        
	FAULT_ACTIVE											:= 2#0000_1000 //2#x0xx_1000 / The Drive is in fault state and awaiting a reset trigger
	
);                                                                          
END_TYPE

// POUs/IO/Drives/SoE/Ax5000ParamSTRUCTs/P/AX5000_P_0001
TYPE AX5000_P_0001 :
STRUCT
	Schwitching_frequencyof_the_IGBT_module:UINT;
END_STRUCT
END_TYPE

// POUs/IO/Drives/SoE/Ax5000ParamSTRUCTs/P/AX5000_P_0002
TYPE AX5000_P_0002 :
STRUCT
	Current_ctrl_cycle_time:UINT:=100;
END_STRUCT
END_TYPE

// POUs/IO/Drives/SoE/Ax5000ParamSTRUCTs/P/AX5000_P_0003
TYPE AX5000_P_0003 :
STRUCT
	Velocity_crtl_cycle_time:UINT;
END_STRUCT
END_TYPE

// POUs/IO/Drives/SoE/Ax5000ParamSTRUCTs/P/AX5000_P_0004
TYPE AX5000_P_0004 :
STRUCT
	Position_ctrl_cycle_time:UINT;
END_STRUCT
END_TYPE

// POUs/IO/Drives/SoE/Ax5000ParamSTRUCTs/P/AX5000_P_0009
TYPE AX5000_P_0009 :
STRUCT
	Synchronisations_mode:UINT;
END_STRUCT
END_TYPE

// POUs/IO/Drives/SoE/Ax5000ParamSTRUCTs/P/AX5000_P_0010
TYPE AX5000_P_0010 :
STRUCT
	Synchronization_mode:ARRAY[0..3] OF UINT;
END_STRUCT
END_TYPE

// POUs/IO/Drives/SoE/Ax5000ParamSTRUCTs/P/AX5000_P_0020
TYPE AX5000_P_0020 :
STRUCT
	EhterCAT_device_identification:UINT:=1;
END_STRUCT
END_TYPE

// POUs/IO/Drives/SoE/Ax5000ParamSTRUCTs/P/AX5000_P_0021
TYPE AX5000_P_0021 :
STRUCT
	Save_EtherCAT_device_identification:UINT;
END_STRUCT
END_TYPE

// POUs/IO/Drives/SoE/Ax5000ParamSTRUCTs/P/AX5000_P_0040
TYPE AX5000_P_0040 :
STRUCT
	ADDitional_drive_status_word:ARRAY[0..14] OF BOOL;
END_STRUCT
END_TYPE

// POUs/IO/Drives/SoE/Ax5000ParamSTRUCTs/P/AX5000_P_0050
TYPE AX5000_P_0050 :
STRUCT
	Funktional_principle:INT;
	Construktion:INT;
	revd:ARRAY[0..14] OF UINT;

END_STRUCT
END_TYPE

// POUs/IO/Drives/SoE/Ax5000ParamSTRUCTs/P/AX5000_P_0051
TYPE AX5000_P_0051 :
STRUCT
	Number_of_pole_pairs:UINT;
END_STRUCT
END_TYPE

// POUs/IO/Drives/SoE/Ax5000ParamSTRUCTs/P/AX5000_P_0052
TYPE AX5000_P_0052 :
STRUCT
	Time_limitation_for_peak_current:UINT;
END_STRUCT
END_TYPE

// POUs/IO/Drives/SoE/Ax5000ParamSTRUCTs/P/AX5000_P_0053
TYPE AX5000_P_0053 :
STRUCT
	Actual_lenght:UINT;
	Max_lenght:UINT;
	Configures_motor_type:STRING(29);

END_STRUCT
END_TYPE

// POUs/IO/Drives/SoE/Ax5000ParamSTRUCTs/P/AX5000_P_0054
TYPE AX5000_P_0054 :
STRUCT
	Actual_lenght:UINT;
	Max_lenght:UINT;
	Configures_drive_type:STRING(29);
END_STRUCT
END_TYPE

// POUs/IO/Drives/SoE/Ax5000ParamSTRUCTs/P/AX5000_P_0055
TYPE AX5000_P_0055 :
STRUCT
	Motor_EMK:WORD;	(*Decimal Point: 1 *)
END_STRUCT
END_TYPE

// POUs/IO/Drives/SoE/Ax5000ParamSTRUCTs/P/AX5000_P_0056
TYPE AX5000_P_0056 :
STRUCT
	Max_motor_speed_with_max_torque:UDINT;
END_STRUCT
END_TYPE

// POUs/IO/Drives/SoE/Ax5000ParamSTRUCTs/P/AX5000_P_0057
TYPE AX5000_P_0057 :
STRUCT
	Electrical_commutation_offset:UINT;
END_STRUCT
END_TYPE

// POUs/IO/Drives/SoE/Ax5000ParamSTRUCTs/P/AX5000_P_0058
TYPE AX5000_P_0058 :
STRUCT
	Mechanical_commutation_offset:UINT;
END_STRUCT
END_TYPE

// POUs/IO/Drives/SoE/Ax5000ParamSTRUCTs/P/AX5000_P_0059
TYPE AX5000_P_0059 :
STRUCT
	Motor_brake_current_monitoring_level:UINT;
END_STRUCT
END_TYPE

// POUs/IO/Drives/SoE/Ax5000ParamSTRUCTs/P/AX5000_P_0060
TYPE AX5000_P_0060 :
STRUCT
	Motor_type_and_usage:WORD;	(* "0"-->no break;standard holding break, "1"-->currentless locked,standard holding break, "16"-->no break; Holding emergency break, "17"-->currentless locked, olding emergency break*)
//	{attribute 'hide'}
	rsvd:ARRAY[0..7] OF UINT;
END_STRUCT
END_TYPE

// POUs/IO/Drives/SoE/Ax5000ParamSTRUCTs/P/AX5000_P_0061
TYPE AX5000_P_0061 :
STRUCT
	Motor_temperature_sensor_type:UINT;
END_STRUCT
END_TYPE

// POUs/IO/Drives/SoE/Ax5000ParamSTRUCTs/P/AX5000_P_0062
TYPE AX5000_P_0062 :
STRUCT
	Actual_lenght:UINT;
	Max_lenght:UINT;
	Time_constant:UINT;
	Warning_limit:UINT;
	Error_limit:UINT;
	Reaktion:UINT;
END_STRUCT
END_TYPE

// POUs/IO/Drives/SoE/Ax5000ParamSTRUCTs/P/AX5000_P_0063
TYPE AX5000_P_0063 :
STRUCT
	Thermal_motor_ulitisation:UINT;
END_STRUCT
END_TYPE

// POUs/IO/Drives/SoE/Ax5000ParamSTRUCTs/P/AX5000_P_0064
TYPE AX5000_P_0064 :
STRUCT
	Actual_motorbrake_current:UINT;
END_STRUCT
END_TYPE

// POUs/IO/Drives/SoE/Ax5000ParamSTRUCTs/P/AX5000_P_0065
TYPE AX5000_P_0065 :
STRUCT
	Actual_temperature_sensor_resistance:UINT;
END_STRUCT
END_TYPE

// POUs/IO/Drives/SoE/Ax5000ParamSTRUCTs/P/AX5000_P_0066
TYPE AX5000_P_0066 :
STRUCT
	Actual_lenght:UINT;
	Max_lenght:UINT;

	iWinding_resistance:UDINT;
	iWinding_inductance:UDINT;
END_STRUCT
END_TYPE

// POUs/IO/Drives/SoE/Ax5000ParamSTRUCTs/P/AX5000_P_0067
TYPE AX5000_P_0067 :
STRUCT
	Motor_winding_dielektric_strength:UINT;
END_STRUCT
END_TYPE

// POUs/IO/Drives/SoE/Ax5000ParamSTRUCTs/P/AX5000_P_0068
TYPE AX5000_P_0068 :
STRUCT
	Actual_lenght:UINT;
	Max_lenght:UINT;
	Overload_factor:UINT;
	CRC16:UINT;
END_STRUCT
END_TYPE

// POUs/IO/Drives/SoE/Ax5000ParamSTRUCTs/P/AX5000_P_0069
TYPE AX5000_P_0069 :
STRUCT
	Actual_lenght:UINT:=2;
	Max_lenght:UINT:=2;
	velocity_limit:UINT:=100;
//	{attribute 'hide'}
	Rsvd:UINT;
END_STRUCT
END_TYPE

// POUs/IO/Drives/SoE/Ax5000ParamSTRUCTs/P/AX5000_P_0070
TYPE AX5000_P_0070 :
STRUCT
	Motor_contunuouse_stall_torque:UINT;
END_STRUCT
END_TYPE

// POUs/IO/Drives/SoE/Ax5000ParamSTRUCTs/P/AX5000_P_0071
TYPE AX5000_P_0071 :
STRUCT
	Actual_lenght:UINT;
	Max_lenght:UINT;
	Rotor_moment_of_inertia:UDINT;
	Load_moment_of_inertia:UDINT;
END_STRUCT
END_TYPE

// POUs/IO/Drives/SoE/Ax5000ParamSTRUCTs/P/AX5000_P_0072
TYPE AX5000_P_0072 :
STRUCT
	Actual_lenght:UINT;
	Max_lenght:UINT;
	Holding_torque:UINT;
	Elektrical_power:UINT;
	Moment_of_inertia:UINT;
END_STRUCT
END_TYPE

// POUs/IO/Drives/SoE/Ax5000ParamSTRUCTs/P/AX5000_P_0073
TYPE AX5000_P_0073 :
STRUCT
	Motor_peak_torque:UDINT;
END_STRUCT
END_TYPE

// POUs/IO/Drives/SoE/Ax5000ParamSTRUCTs/P/AX5000_P_0074
TYPE AX5000_P_0074 :
STRUCT
	Actual_lenght:UINT;
	Max_lenght:UINT;
	Iq: ARRAY [0..9] OF UDINT;
	M: ARRAY [0..9] OF UDINT;
END_STRUCT
END_TYPE

// POUs/IO/Drives/SoE/Ax5000ParamSTRUCTs/P/AX5000_P_0075
TYPE AX5000_P_0075 :
STRUCT
	Actual_lenght:UINT;
	Max_lenght:UINT;
	Iq: ARRAY[0..9] OF UDINT;
	Lq:ARRAY[0..9] OF UDINT;
END_STRUCT
END_TYPE

// POUs/IO/Drives/SoE/Ax5000ParamSTRUCTs/P/AX5000_P_0076
TYPE AX5000_P_0076 :
STRUCT
	Actual_lenght:UINT;
	Max_lenght:UINT;
	Temperature:ARRAY [0..9] OF UINT;
	Resistance:ARRAY [0..9] OF UINT;
END_STRUCT
END_TYPE

// POUs/IO/Drives/SoE/Ax5000ParamSTRUCTs/P/AX5000_P_0077
TYPE AX5000_P_0077 :
STRUCT
	Motor_rated_voltage:UINT;
END_STRUCT
END_TYPE

// POUs/IO/Drives/SoE/Ax5000ParamSTRUCTs/P/AX5000_P_0078
TYPE AX5000_P_0078 :
STRUCT
	Max_motor_dc_link_voltage:UINT;
END_STRUCT
END_TYPE

// POUs/IO/Drives/SoE/Ax5000ParamSTRUCTs/P/AX5000_P_0088
TYPE AX5000_P_0088 :
STRUCT
	Velocity_limit_value:UDINT;
	Corresponding_current_value:UINT;
END_STRUCT
END_TYPE

// POUs/IO/Drives/SoE/Ax5000ParamSTRUCTs/P/AX5000_P_0089
TYPE AX5000_P_0089 :
STRUCT
	Actual_lenght:UINT;
	Max_lenght:UINT;
	IDN:UDINT;
	MinValue:UDINT;
	MaxValue:UDINT;
	IDN2:UDINT;
	MinValue2:UDINT;
	MaxValue2:UDINT;
	IDN3:UDINT;
	MinValue3:UDINT;
	MaxValue3:UDINT;
END_STRUCT
END_TYPE

// POUs/IO/Drives/SoE/Ax5000ParamSTRUCTs/P/AX5000_P_0090
TYPE AX5000_P_0090 :
STRUCT
	Channel_peak_current:UDINT;
END_STRUCT
END_TYPE

// POUs/IO/Drives/SoE/Ax5000ParamSTRUCTs/P/AX5000_P_0091
TYPE AX5000_P_0091 :
STRUCT
	Channel_rated_current:UDINT;
END_STRUCT
END_TYPE

// POUs/IO/Drives/SoE/Ax5000ParamSTRUCTs/P/AX5000_P_0092
TYPE AX5000_P_0092 :
STRUCT
	Configured_channel_peak_current:UDINT;
END_STRUCT
END_TYPE

// POUs/IO/Drives/SoE/Ax5000ParamSTRUCTs/P/AX5000_P_0093
TYPE AX5000_P_0093 :
STRUCT
	Configures_channel_current:UDINT;
END_STRUCT
END_TYPE

// POUs/IO/Drives/SoE/Ax5000ParamSTRUCTs/P/AX5000_P_0096
TYPE AX5000_P_0096 :
STRUCT
	Motor_brake_force_lock:BOOL;
	Motor_brake_force_unlock:BOOL;
//	{attribute 'hide'}
	Rsvd:ARRAY[0..13] OF BOOL;
END_STRUCT
END_TYPE

// POUs/IO/Drives/SoE/Ax5000ParamSTRUCTs/P/AX5000_P_0097
TYPE AX5000_P_0097 :
STRUCT
	Motor_break_unlocked:BOOL;
	Rsvd:ARRAY[0..14] OF BOOL;
END_STRUCT
END_TYPE

// POUs/IO/Drives/SoE/Ax5000ParamSTRUCTs/P/AX5000_P_0098_beckhoff
{attribute 'pack_mode' := '1'} //Ensures 1-byte-alignmend
TYPE AX5000_P_0098_beckhoff :
STRUCT
	Actual_lenght : UINT := 16#80;
	Max_lenght : UINT := 16#80;
	Name_plate_type: E_AX5000_P_0150_DigitalNamePlate;
//	{attribute 'hide'}
	Rsvd1:ARRAY[0..0] OF UINT;
	Id_prat_1:UDINT;
	Id_prat_2:UDINT;
	Version_no:UINT;
	Motor_vendor:UINT;
	Serial_number:UDINT;
	Motor_type:STRING(29);
	Feedback_typ:STRING(29);
//	{attribute 'hide'}
	Rsvd2:UINT;
	Add_motor_parameter_description:UINT;
	Nominal_current:UDINT;
	Nominal_voltage:UINT;
	Nominal_frequenz:UINT;
	Nominal_speed:UINT;
	Maximun_speed:UINT;
	Cos_phi:UINT;
	Maximum_feedback_speed:UINT;
//	{attribute 'hide'}
	Rsvd3:ARRAY[0..5] OF UINT;	
//	{attribute 'hide'}
	Rsvd4:UINT;
	Checksum:UINT;
	Position_offset:UDINT;
	Number_of_adjustments:UINT;
	
	Additional_mech_position_offset:UDINT;
	Checksum2:UINT;
(*
	Vendor:STRING(29);
	Order_code:STRING(29);
	Electric_type:STRING(29);
	Serial_no:STRING(10);
	 {attribute 'hide'}
	rsvd5:ARRAY[0..9] OF UINT;
	Mechanical_commutation_offset:UDINT;
	Generic:ARRAY[0..61] OF UINT;*)
END_STRUCT
END_TYPE

// POUs/IO/Drives/SoE/Ax5000ParamSTRUCTs/P/AX5000_P_0098_beckhoff_electrical_data
{attribute 'pack_mode' := '1'}//Ensures 1-byte-alignmend
TYPE AX5000_P_0098_beckhoff_electrical_data :
STRUCT
	Actual_lenght:UINT;
	Max_lenght:UINT;
	Name_plate_type:UINT;
//	 {attribute 'hide'}
	Rsvd1:ARRAY[0..0] OF UINT;
	(*Id_prat_1:UDINT;
	Id_prat_2:UDINT;
	Version_no:UINT;
	Motor_vendor:UINT;
	Serial_number:UDINT;
	Motor_type:STRING(29);
	Feedback_typ:STRING(29);
	 {attribute 'hide'}
	rsvd2:UINT;
	Add_motor_parameter_description:UINT;
	Nominal_current:UDINT;
	Nominal_voltage:UINT;
	Nominal_frequenz:UINT;
	Nominal_speed:UINT;
	Maximun_speed:UINT;
	Cos_phi:UINT;
	Maximum_feedback_speed:UINT;
	 {attribute 'hide'}
	Rsvd3:ARRAY[0..5] OF UINT;
	Checksum:UINT;
	Position_offset:UDINT;
	Number_of_adjustments:UINT;
	Additional_mech_position_offset:UDINT;
	Checksum2:UINT;*)

	Vendor:STRING(29);
	Order_code:STRING(29);
	Electric_type:STRING(29);
	Serial_no:STRING(9);
//	{attribute 'hide'}
	Rsvd5:ARRAY[0..9] OF UINT;
	Mechanical_commutation_offset:UDINT;
	(*Generic:ARRAY[0..61] OF UINT;*)
END_STRUCT
END_TYPE

// POUs/IO/Drives/SoE/Ax5000ParamSTRUCTs/P/AX5000_P_0099
{attribute 'pack_mode' := '1'}//Ensures 1-byte-alignmend
TYPE AX5000_P_0099 :
STRUCT
	Actual_lenght:UINT;
	Max_lenght:UINT;
	Request:UINT;
	Encoder_connector:UINT;
	File:UINT;
	File_size_in_words:UINT;
//	{attribute 'hide'}
	Rsvd:ARRAY [0..1] OF UINT;
	Offset_in_Words:UINT;
	Length_in_words:UINT;
	Response:UINT;
	Data_state:UINT;
	File_size_in_words2:UINT;
//	{attribute 'hide'}
	Rsvd1:UINT;
//	{attribute 'hide'}
	Rsvd2: UDINT;
	Offset_in_words2:UINT;
	Length_in_words2:UINT;
	Data_array:ARRAY[0..255] OF UINT;

END_STRUCT
END_TYPE

// POUs/IO/Drives/SoE/Ax5000ParamSTRUCTs/P/AX5000_P_0100
TYPE AX5000_P_0100 :
STRUCT
	ASM_nominal_speed:UDINT;
END_STRUCT
END_TYPE

// POUs/IO/Drives/SoE/Ax5000ParamSTRUCTs/P/AX5000_P_0101
TYPE AX5000_P_0101 :
STRUCT
	ASM_nominal_voltage:UINT;
END_STRUCT
END_TYPE

// POUs/IO/Drives/SoE/Ax5000ParamSTRUCTs/P/AX5000_P_0102
TYPE AX5000_P_0102 :
STRUCT
	ASM_nominal_frequency:UINT;
END_STRUCT
END_TYPE

// POUs/IO/Drives/SoE/Ax5000ParamSTRUCTs/P/AX5000_P_0103
TYPE AX5000_P_0103 :
STRUCT
	ASM_boost_voltage:UINT;
END_STRUCT
END_TYPE

// POUs/IO/Drives/SoE/Ax5000ParamSTRUCTs/P/AX5000_P_0104
TYPE AX5000_P_0104 :
STRUCT
	ASM_power_faktor:UINT;
END_STRUCT
END_TYPE

// POUs/IO/Drives/SoE/Ax5000ParamSTRUCTs/P/AX5000_P_0105
TYPE AX5000_P_0105 :
STRUCT
	ASM_Rotor_time_constant:UINT;
END_STRUCT
END_TYPE

// POUs/IO/Drives/SoE/Ax5000ParamSTRUCTs/P/AX5000_P_0106
TYPE AX5000_P_0106 :
STRUCT
	ASM_connection_type:UINT;
END_STRUCT
END_TYPE

// POUs/IO/Drives/SoE/Ax5000ParamSTRUCTs/P/AX5000_P_0107
TYPE AX5000_P_0107 :
STRUCT
	ASM_Magnetizing_current:UDINT;
END_STRUCT
END_TYPE

// POUs/IO/Drives/SoE/Ax5000ParamSTRUCTs/P/AX5000_P_0108
TYPE AX5000_P_0108 :
STRUCT
	ASM_stator_resistance:UDINT;
END_STRUCT
END_TYPE

// POUs/IO/Drives/SoE/Ax5000ParamSTRUCTs/P/AX5000_P_0109
TYPE AX5000_P_0109 :
STRUCT
	ASM_stator_leakage_inductance:UDINT;
END_STRUCT
END_TYPE

// POUs/IO/Drives/SoE/Ax5000ParamSTRUCTs/P/AX5000_P_0110
TYPE AX5000_P_0110 :
STRUCT
	ASM_motor_magnetzing_inductance:UDINT;
END_STRUCT
END_TYPE

// POUs/IO/Drives/SoE/Ax5000ParamSTRUCTs/P/AX5000_P_0111
TYPE AX5000_P_0111 :
STRUCT
	ASM_rotor_leakage_inductance:UDINT;
END_STRUCT
END_TYPE

// POUs/IO/Drives/SoE/Ax5000ParamSTRUCTs/P/AX5000_P_0112
TYPE AX5000_P_0112 :
STRUCT
	ASM_acceleration_control_torque_limit_value:UINT;
END_STRUCT
END_TYPE

// POUs/IO/Drives/SoE/Ax5000ParamSTRUCTs/P/AX5000_P_0113
TYPE AX5000_P_0113 :
STRUCT
	ASM_acceleration_control_proportional_gain:UDINT;
END_STRUCT
END_TYPE

// POUs/IO/Drives/SoE/Ax5000ParamSTRUCTs/P/AX5000_P_0114
TYPE AX5000_P_0114 :
STRUCT
	ASM_acceleration_control_integral_action_time:UINT;
END_STRUCT
END_TYPE

// POUs/IO/Drives/SoE/Ax5000ParamSTRUCTs/P/AX5000_P_0115
TYPE AX5000_P_0115 :
STRUCT
	ASM_stall_protection_loop_torque_limit_value:UINT;
END_STRUCT
END_TYPE

// POUs/IO/Drives/SoE/Ax5000ParamSTRUCTs/P/AX5000_P_0116
TYPE AX5000_P_0116 :
STRUCT
	ASM_stall_protection_loop_proportional_gain:UDINT;
END_STRUCT
END_TYPE

// POUs/IO/Drives/SoE/Ax5000ParamSTRUCTs/P/AX5000_P_0117
TYPE AX5000_P_0117 :
STRUCT
	ASM_stall_protection_loop_intrgral_action_time:UINT;
END_STRUCT
END_TYPE

// POUs/IO/Drives/SoE/Ax5000ParamSTRUCTs/P/AX5000_P_0118
TYPE AX5000_P_0118 :
STRUCT
	ASM_slip_compension_factor:UINT;
END_STRUCT
END_TYPE

// POUs/IO/Drives/SoE/Ax5000ParamSTRUCTs/P/AX5000_P_0119
TYPE AX5000_P_0119 :
STRUCT
	ASM_boost_voltage_slope:UDINT;
END_STRUCT
END_TYPE

// POUs/IO/Drives/SoE/Ax5000ParamSTRUCTs/P/AX5000_P_0125
TYPE AX5000_P_0125 :
STRUCT
	Pole_pair_distance:UINT;
END_STRUCT
END_TYPE

// POUs/IO/Drives/SoE/Ax5000ParamSTRUCTs/P/AX5000_P_0126
TYPE AX5000_P_0126 :
STRUCT
	Motor_continouse_stall_force:UDINT;
END_STRUCT
END_TYPE

// POUs/IO/Drives/SoE/Ax5000ParamSTRUCTs/P/AX5000_P_0127
TYPE AX5000_P_0127 :
STRUCT
	Actual_lenght:UINT;
	Max_lenght:UINT;
	Coil_unit_mass:UDINT;
	Load_mass:UDINT;
END_STRUCT
END_TYPE

// POUs/IO/Drives/SoE/Ax5000ParamSTRUCTs/P/AX5000_P_0128
TYPE AX5000_P_0128 :
STRUCT
	Motor_peak_force:UDINT;
END_STRUCT
END_TYPE

// POUs/IO/Drives/SoE/Ax5000ParamSTRUCTs/P/AX5000_P_0150
TYPE AX5000_P_0150 EXTENDS ST_AX5000_P_0150 :
STRUCT
(*
	Actual_lenght:UINT:=224;
	Max_lenght:UINT:=224;

	Manufacturer:UINT:=2;
	Feedback_type:UINT:=1;
	Feedback_type_string:STRING(29):='hallo';
	Feedback_use:UINT:=3;
	Feedback_direction:UINT:=1;
//{attribute 'hide'}
	Rsvd1:ARRAY[0..2] OF UINT;

	(*Powersettlings*)
	Control_voltage:UINT;
	Wait_time_after_power_up:UINT;
	Connector:UINT;
//	{attribute 'hide'}	
	Rsvd2:ARRAY[0..2] OF UINT;

	(*Process channel*)
		Process_interface:UINT;
		Conector2:UINT;
			(*rsvd*)
			// {attribute 'hide'}
				Rsvd3:ARRAY[0..1] OF UINT;
			(*Data*)
				(*Sin/Cos*)
					Resulution_per_rotation:UDINT;
					Length_per_signal_period:UDINT;
					Sin_gain_correction:UINT;
					Sin_offset_correction:UINT;
					Cos_gain_correction:UINT;
					Cos_offset_correction:UINT;
					Sin_Cos_1Vss_monitoring:UINT;
					// {attribute 'hide'}
					Rsvd4:ARRAY[0..10] OF UINT;
				(*TTL*)
					(*Resolution_per_rotation:UDINT;
					Length_per_signal_period:UDINT;
					rsvd5:ARRAY[0..15] OF UINT;*)
				(*Resolver*)
					(*Control_word:UINT;
					Number_of_poles:USINT;
					Exibition_frequency:USINT;
					Transformation_ratio:UINT;
					Phase_shift:UINT;
					Sin_cos_amplitude_monitoring:UINT;
						 {attribute 'hide'}
					rsvd6:UINT;
					Amplitude_monitoring_max_limit:UINT;
					Amplitude_monitoring_min_limit:UINT;
					Observer_bandwidth:UINT;
					Observer_correction_factor_Iq_to_acc:UINT;
						 {attribute 'hide'}
					rsvd7:ARRAY[0..4] OF UDINT;*)
				(*MES*)
					(*Control_word:UINT;
						 {attribute 'hide'}
					rsvd8:UINT;
					sin_offset:UINT;
					cos_offset:UINT;
					Sin_cos_Amplitude_correction:UINT;
						 {attribute 'hide'}
					rsvd9:UINT;
					Amplitude_monitoring_max_limit:UINT;
					Amplitude_monitoring_min_limit:UINT;
					Observer_bandwidth:UINT;
					Observer_correction_factor_Iq_to_acc:UINT;
						 {attribute 'hide'}
					rsvd10:ARRAY[0..4] OF UDINT;*)
				(*HTL*)
					(*Resulution_per_rotation:UDINT;
					Length_per_signal_period:UDINT;
						 {attribute 'hide'}
					rsvd11:ARRAY[0..15] OF UINT;*)
	(*Parameter channel*)
		Parameter_interface:UINT;
		Conector3:UINT;
		Identifier:UDINT;
		Bit_resolution_singelturn_position:UINT;
		Bit_resolution_multiturn_position:UINT;
		Number_of_clockcycles_to_get_singelturn_position:UINT;
		Number_of_clockcycles_to_get_multiturn_position:UINT;
		Digital_name_plate:UINT;
		commutation_mode_adjustable_commutation_offset:UINT;
		Linear_resolution_about_digital_interface_in_nm:UDINT;
		//	 {attribute 'hide'}
		Rsvd12:ARRAY[0..3] OF UINT;
		data:ARRAY[0..29] OF UINT;
	(*manufacturer limits settings*)
		Maximum_continous_operation_speed:UINT;
		Maximum_continous_mechenical_speed:UINT;
		Maximum_temperature:UINT;
		//	 {attribute 'hide'}
		Rsvd13:ARRAY[0..2] OF UINT;

	FeedbackOption :UDINT:=1;
	//	 {attribute 'hide'}
	Reserve :ARRAY[0..5] OF UINT;

*)
END_STRUCT
END_TYPE

// POUs/IO/Drives/SoE/Ax5000ParamSTRUCTs/P/AX5000_P_0151
{attribute 'pack_mode' := '1'}//Ensures 1-byte-alignmend
TYPE AX5000_P_0151 :
STRUCT
	Actual_lenght:UINT;
	Max_lenght:UINT;
	Manufacturer:UINT;
	Feedback_type:UINT;
	Feedback_type_string:STRING(29);
//{attribute 'hide'}
	Rsvd1:ARRAY[0..4] OF UINT;
	Process_channel:ARRAY[0..11] OF UINT;
	Parameter_channel:ARRAY[0..77] OF UINT;
	Manufacturer_limits_settings:ARRAY[0..5] OF UINT;
//{attribute 'hide'}
	Rsvd2:ARRAY[0..7] OF UINT;
END_STRUCT
END_TYPE

// POUs/IO/Drives/SoE/Ax5000ParamSTRUCTs/P/AX5000_P_0152
TYPE AX5000_P_0152 :
STRUCT
	Feedback_1_geat_numerator:UDINT;
END_STRUCT
END_TYPE

// POUs/IO/Drives/SoE/Ax5000ParamSTRUCTs/P/AX5000_P_0153
TYPE AX5000_P_0153 :
STRUCT
	Feedback_1_geat_denominator:UDINT;
END_STRUCT
END_TYPE

// POUs/IO/Drives/SoE/Ax5000ParamSTRUCTs/P/AX5000_P_0154
TYPE AX5000_P_0154 :
STRUCT
	Actual_lenght:UINT;
	Max_lenght:UINT;
	Reference_source:UINT;
	Reference_index:UINT;
	Threshold_voltage:UINT;
//{attribute 'hide'}
	rsvd:UINT;
END_STRUCT
END_TYPE

// POUs/IO/Drives/SoE/Ax5000ParamSTRUCTs/P/AX5000_P_0155
TYPE AX5000_P_0155 :
STRUCT
	Feedback_1_resolution_scaling:UDINT;
END_STRUCT
END_TYPE

// POUs/IO/Drives/SoE/Ax5000ParamSTRUCTs/P/AX5000_P_0158
TYPE AX5000_P_0158 :
STRUCT
	Save_feedback_identication:UINT;
END_STRUCT
END_TYPE

// POUs/IO/Drives/SoE/Ax5000ParamSTRUCTs/P/AX5000_P_0159
TYPE AX5000_P_0159 :
STRUCT
	Raw_position_feedback_value:UDINT;
END_STRUCT
END_TYPE

// POUs/IO/Drives/SoE/Ax5000ParamSTRUCTs/P/AX5000_P_0160
TYPE AX5000_P_0160 :
STRUCT
	Calibrate_commutation_offset:UINT;
END_STRUCT
END_TYPE

// POUs/IO/Drives/SoE/Ax5000ParamSTRUCTs/P/AX5000_P_0161
TYPE AX5000_P_0161 :
STRUCT
	Feedback1_save_commutation_offset:UINT;
END_STRUCT
END_TYPE

// POUs/IO/Drives/SoE/Ax5000ParamSTRUCTs/P/AX5000_P_0162
TYPE AX5000_P_0162 :
STRUCT
	Feedback1_save_digital_nameplate:UINT;
END_STRUCT
END_TYPE

// POUs/IO/Drives/SoE/Ax5000ParamSTRUCTs/P/AX5000_P_0163
TYPE AX5000_P_0163 :
STRUCT
	Scan_feedback1:UINT;
END_STRUCT
END_TYPE

// POUs/IO/Drives/SoE/Ax5000ParamSTRUCTs/P/AX5000_P_0165
{attribute 'pack_mode' := '1'}//Ensures 1-byte-alignmend
TYPE AX5000_P_0165 :
STRUCT
	Actual_lenght:UINT;
	Max_lenght:UINT;
	Command_mode:UINT;
	Activation:UINT;
	
//{attribute 'hide'}
	Rsvd1:ARRAY[0..1] OF UINT;
	Current_level:UINT;
	Duration:UINT;
//{attribute 'hide'}
	Rsvd2:ARRAY[0..3] OF UINT;
	First_phase_current_level:UINT;
	First_phase_ramp_up_time:UINT;
	Second_phase_current_level:UINT;
	Second_phase_ramp_up_time:UINT;
	Commutation_pos_control_Kp:UINT;
	First_phase_pos_monitoring_limit:UINT;
	First_phase_step_width:UINT;
	First_phase_wating_time_after_step:UINT;
	Second_phase_duration:UINT;
	Error_monitoring:UINT;
//{attribute 'hide'}
	Rsvd3:ARRAY[0..9] OF UINT;


END_STRUCT
END_TYPE

// POUs/IO/Drives/SoE/Ax5000ParamSTRUCTs/P/AX5000_P_0166
TYPE AX5000_P_0166 :
STRUCT
	Motor_and_feedback_connection_ceck:UINT;
END_STRUCT
END_TYPE

// POUs/IO/Drives/SoE/Ax5000ParamSTRUCTs/P/AX5000_P_0167
{attribute 'pack_mode' := '1'}//Ensures 1-byte-alignmend
TYPE AX5000_P_0167 :
STRUCT
	Actual_lenght:UINT;
	Max_lenght:UINT;
	eMode:UINT;
	Current_level:UINT;
	Moving_distance:UINT;
	Velocety:UINT;
//{attribute 'hide'}
	Rsvd:UINT;
//{attribute 'hide'}
	Rsvd2:UINT;
	EqualDirektions:UINT;
	Commutation_position_difference:UINT;
//{attribute 'hide'}
	Rsvd3:UINT;
//{attribute 'hide'}
	Rsvd4:UINT;

END_STRUCT
END_TYPE

// POUs/IO/Drives/SoE/Ax5000ParamSTRUCTs/P/AX5000_P_0168
{attribute 'pack_mode' := '1'}//Ensures 1-byte-alignmend
TYPE AX5000_P_0168 :
STRUCT
	Actual_lenght:UINT;
	Max_lenght:UINT;
	Phase_shift:UINT;
	Sin_offset_correction:UINT;
	Cos_offset_correction:UINT;
//{attribute 'hide'}
	Rsvd:ARRAY[0..6] OF UINT;
	Vector_length:UINT;
	Sin_max:UINT;
	Sin_min:UINT;
	Cos_max:UINT;
	Cos_min:UINT;
//{attribute 'hide'}
	Rsvd2:ARRAY[0..4] OF UINT;

END_STRUCT
END_TYPE

// POUs/IO/Drives/SoE/Ax5000ParamSTRUCTs/P/AX5000_P_0169
{attribute 'pack_mode' := '1'}//Ensures 1-byte-alignmend
TYPE AX5000_P_0169 :
STRUCT
	Actual_lenght:UINT;
	Max_lenght:UINT;
(*Onboard*)
	DelayRegister:UINT;
	QualityMonitorValue:UINT;
	SlaveRSSI:UINT;
	EdgeRegister:UINT;
	SummaryRegister:UINT;
	EncoderTemperature:INT;
	LEDCurrent:UINT;
	SupplyVoltage:UINT;
	EncoderStatus0:USINT;
	EncoderStatus1:USINT;
	EncoderStatus2:USINT;
	EncoderStatus3:USINT;
	EncoderStatus4:USINT;
	EncoderStatus5:USINT;
	EncoderStatus6:USINT;
	EncoderStatus7:USINT;
	EncoderStatus0_detailed:USINT;
	EncoderStatus1_detailed:USINT;
	EncoderStatus2_detailed:USINT;
	EncoderStatus3_detailed:USINT;
	EncoderStatus4_detailed:USINT;
	EncoderStatus5_detailed:USINT;
	EncoderStatus6_detailed:USINT;
	EncoderStatus7_detailed:USINT;
	OperatingTime:UDINT;
	TotalShaftTurns:UDINT;
//{attribute 'hide'}
	Rsvd:ARRAY[0..2] OF UINT;
	MaxOccuredPositionDelivation:UINT;
	TotalVPOSErrors:UINT;
	TotalACCErrors:UINT;
	TotalPOSErrors:UINT;
	TotalLINKErrors:UINT;
	TotalEncodingErrors:UINT;
//{attribute 'hide'}
	Rsvd2:UINT;
//{attribute 'hide'}
	Rsvd3:UINT;
	CyclicReadCounter:UINT;
	CyclicReadErrorCounter:UINT;


(*AX57xx*)			(*Die beiden NICHT verwendeten Feedbacksystemeauf der AX57xx müssen ausgeklammert werden*)

		(*HiperfaceDSL
			DelayRegister:UINT;
			QualityMonitorValue:UINT;
			SlaveRSSI:UINT;
			EdgeRegister:UINT;
			SummaryRegister:UINT;
			EncoderTemperature:INT;
			LEDCurrent:UINT;
			SupplyVoltage:UINT;
			EncoderStatus0:USINT;
			EncoderStatus1:USINT;
			EncoderStatus2:USINT;
			EncoderStatus3:USINT;
			EncoderStatus4:USINT;
			EncoderStatus5:USINT;
			EncoderStatus6:USINT;
			EncoderStatus7:USINT;
			EncoderStatus0_detailed:USINT;
			EncoderStatus1_detailed:USINT;
			EncoderStatus2_detailed:USINT;
			EncoderStatus3_detailed:USINT;
			EncoderStatus4_detailed:USINT;
			EncoderStatus5_detailed:USINT;
			EncoderStatus6_detailed:USINT;
			EncoderStatus7_detailed:USINT;
			OperatingTime:UDINT;
			TotalShaftTurns:UDINT;
	//	{attribute 'hide'}
			rsvd:ARRAY[0..2] OF UINT;
			MaxOccuredPositionDelivation:UINT;
			TotalVPOSErrors:UINT;
			TotalACCErrors:UINT;
			TotalPOSErrors:UINT;
			TotalLINKErrors:UINT;
			TotalEncodingErrors:UINT;
		//	{attribute 'hide'}
			rsvd2:UINT;
		//	{attribute 'hide'}
			rsvd3:UINT;
			CyclicReadCounter:UINT;
			CyclicReadErrorCounter:UINT;
*)
(*

		(*AX572xEnDat2.2*)

			AX572xEnDat2.2:UINT;

*)

(*
		(*AX572xBiSS*)

			AX572xBiSS:UINT;
*)

END_STRUCT
END_TYPE

// POUs/IO/Drives/SoE/Ax5000ParamSTRUCTs/P/AX5000_P_0170
TYPE AX5000_P_0170 :
STRUCT
	Feedback_data_state:UINT;
END_STRUCT
END_TYPE

// POUs/IO/Drives/SoE/Ax5000ParamSTRUCTs/P/AX5000_P_0171
{attribute 'pack_mode' := '1'}//Ensures 1-byte-alignmend
TYPE AX5000_P_0171 :
STRUCT
	Actual_lenght:UINT;
	Max_lenght:UINT;
	Numeration:UDINT;
	Denominator:UDINT;
	Mask:UDINT;
	Position_offset:UDINT;
	Data_valid:UINT;
//{attribute 'hide'}
	Rsvd:UINT;
END_STRUCT
END_TYPE

// POUs/IO/Drives/SoE/Ax5000ParamSTRUCTs/P/AX5000_P_0180
TYPE AX5000_P_0180 EXTENDS ST_AX5000_P_0180:
STRUCT
(*	Actual_lenght:UINT:=224;
	Max_lenght:UINT:=224;

	Manufacturer:UINT:=2;
	Feedback_type:UINT:=1;
	Feedback_type_string:STRING(29):='';
	Feedback_use:UINT:=3;
	Feedback_direction:UINT:=1;
	(*rsvd*)
//{attribute 'hide'}
		rsvd1:ARRAY[0..2] OF UINT;

	(*Powersettlings*)
		Control_voltage:UINT;
		Wait_time_after_power_up:UINT;
		Connector:UINT;
//	{attribute 'hide'}
		Rsvd2:ARRAY[0..2] OF UINT;

	(*Process channel*)
		Process_interface:UINT;
		Conector2:UINT;
			(*rsvd*)
		//	{attribute 'hide'}
				Rsvd3:ARRAY[0..1] OF UINT;
			(*Data*)
				(*Sin/Cos*)
					Resulution_per_rotation:UDINT;
					Length_per_signal_period:UDINT;
					Sin_gain_correction:UINT;
					Sin_offset_correction:UINT;
					Cos_gain_correction:UINT;
					Cos_offset_correction:UINT;
					Sin_Cos_1Vss_monitoring:UINT;
					Rsvd4:ARRAY[0..10] OF UINT;
				(*TTL*)
					(*Resolution_per_rotation:UDINT;
					Length_per_signal_period:UDINT;
				//	{attribute 'hide'}
					rsvd5:ARRAY[0..15] OF UINT;*)
				(*Resolver*)
					(*Control_word:UINT;
					Number_of_poles:USINT;
					Exibition_frequency:USINT;
					Transformation_ratio:UINT;
					Phase_shift:UINT;
					Sin_cos_amplitude_monitoring:UINT;
				//	{attribute 'hide'}
					rsvd6:UINT;
					Amplitude_monitoring_max_limit:UINT;
					Amplitude_monitoring_min_limit:UINT;
					Observer_bandwidth:UINT;
					Observer_correction_factor_Iq_to_acc:UINT;
					rsvd7:ARRAY[0..4] OF UDINT;*)
				(*MES*)
					(*Control_word:UINT;
				//	{attribute 'hide'}
					rsvd8:UINT;
					sin_offset:UINT;
					cos_offset:UINT;
					Sin_cos_Amplitude_correction:UINT;
					rsvd9:UINT;
					Amplitude_monitoring_max_limit:UINT;
					Amplitude_monitoring_min_limit:UINT;
					Observer_bandwidth:UINT;
					Observer_correction_factor_Iq_to_acc:UINT;
				//	{attribute 'hide'}
					rsvd10:ARRAY[0..4] OF UDINT;*)
				(*HTL*)
					(*Resulution_per_rotation:UDINT;
					Length_per_signal_period:UDINT;
					rsvd11:ARRAY[0..15] OF UINT;*)
	(*Parameter channel*)
		Parameter_interface:UINT;
		Conector3:UINT;
		Identifier:UDINT;
		Bit_resolution_singelturn_position:UINT;
		Bit_resolution_multiturn_position:UINT;
		Number_of_clockcycles_to_get_singelturn_position:UINT;
		Number_of_clockcycles_to_get_multiturn_position:UINT;
		Digital_name_plate:UINT;
		commutation_mode_adjustable_commutation_offset:UINT;
		Linear_reselution_about_digital_interface_in_nm:UDINT;
	//	{attribute 'hide'}
		Rsvd12:ARRAY[0..3] OF UINT;
		Data:ARRAY[0..29] OF UINT;
	(*manufacturer limits settings*)
		Maximum_continous_operation_speed:UINT;
		Maximum_continous_mechenical_speed:UINT;
		Maximum_temperature:UINT;
	//	{attribute 'hide'}
		Rsvd13:ARRAY[0..2] OF UINT;

	FeedbackOption :UDINT:=1;
//	{attribute 'hide'}
	Rsvd14 :ARRAY[0..5] OF UINT;
*)
END_STRUCT
END_TYPE

// POUs/IO/Drives/SoE/Ax5000ParamSTRUCTs/P/AX5000_P_0181
{attribute 'pack_mode' := '1'}//Ensures 1-byte-alignmend
TYPE AX5000_P_0181 :
STRUCT
	Actual_lenght:UINT;
	Max_lenght:UINT;
	Manufacturer:UINT;
	Feedback_type:UINT;
	Feedback_type_string:STRING(29);
//	{attribute 'hide'}
	Rsvd1:ARRAY[0..4] OF UINT;
	Process_channel:ARRAY[0..11] OF UINT;
	Parameter_channel:ARRAY[0..77] OF UINT;
	Manufacturer_limits_settings:ARRAY[0..5] OF UINT;
//	{attribute 'hide'}
	Rsvd2:ARRAY[0..7] OF UINT;
END_STRUCT
END_TYPE

// POUs/IO/Drives/SoE/Ax5000ParamSTRUCTs/P/AX5000_P_0182
TYPE AX5000_P_0182 :
STRUCT
	Feedback_2_geat_numerator:UDINT;
END_STRUCT
END_TYPE

// POUs/IO/Drives/SoE/Ax5000ParamSTRUCTs/P/AX5000_P_0183
TYPE AX5000_P_0183 :
STRUCT
	Feedback_2_geat_denominator:UDINT;
END_STRUCT
END_TYPE

// POUs/IO/Drives/SoE/Ax5000ParamSTRUCTs/P/AX5000_P_0184
{attribute 'pack_mode' := '1'}//Ensures 1-byte-alignmend
TYPE AX5000_P_0184 :
STRUCT
	Actual_lenght:UINT;
	Max_lenght:UINT;
	Reference_source:UINT;
	Reference_index:UINT;
	Threshold_voltage:UINT;
//	{attribute 'hide'}
	Rsvd:UINT;
END_STRUCT
END_TYPE

// POUs/IO/Drives/SoE/Ax5000ParamSTRUCTs/P/AX5000_P_0185
TYPE AX5000_P_0185 :
STRUCT
	Feedback_2_resolution_scaling:UDINT;
END_STRUCT
END_TYPE

// POUs/IO/Drives/SoE/Ax5000ParamSTRUCTs/P/AX5000_P_0188
TYPE AX5000_P_0188 :
STRUCT
	Save_feedback_identication:UINT;
END_STRUCT
END_TYPE

// POUs/IO/Drives/SoE/Ax5000ParamSTRUCTs/P/AX5000_P_0189
TYPE AX5000_P_0189 :
STRUCT
	Raw_position_feedback_value:UDINT;
END_STRUCT
END_TYPE

// POUs/IO/Drives/SoE/Ax5000ParamSTRUCTs/P/AX5000_P_0192
TYPE AX5000_P_0192 :
STRUCT
	Feedback2_save_digital_nameplate:UINT;
END_STRUCT
END_TYPE

// POUs/IO/Drives/SoE/Ax5000ParamSTRUCTs/P/AX5000_P_0193
TYPE AX5000_P_0193 :
STRUCT
	Scan_feedback2:UINT;
END_STRUCT
END_TYPE

// POUs/IO/Drives/SoE/Ax5000ParamSTRUCTs/P/AX5000_P_0196
TYPE AX5000_P_0196 :
STRUCT
	Actual_lenght:UINT;
	Max_lenght:UINT;
	Numeration:UDINT;
	Denominator:UDINT;
	Mask:UDINT;
	Position_offset:UDINT;
	Data_valid:UINT;
//	{attribute 'hide'}
	rsvd:UINT;
END_STRUCT
END_TYPE

// POUs/IO/Drives/SoE/Ax5000ParamSTRUCTs/P/AX5000_P_0198
{attribute 'pack_mode' := '1'}//Ensures 1-byte-alignmend
TYPE AX5000_P_0198 :
STRUCT
	Actual_lenght:UINT;
	Max_lenght:UINT;
	Feedback_instance:UINT;
	Cmd:UINT;
	Timeout:UINT;
	Byte_length:UINT;
	Addr:UDINT;
	Byte2_length:UINT;
	Error_code_as_response:UINT;
	Data: ARRAY [0..3] OF UINT;
END_STRUCT
END_TYPE

// POUs/IO/Drives/SoE/Ax5000ParamSTRUCTs/P/AX5000_P_0199
TYPE AX5000_P_0199 :
STRUCT
	Direct_feedback_access:UINT;
END_STRUCT
END_TYPE

// POUs/IO/Drives/SoE/Ax5000ParamSTRUCTs/P/AX5000_P_0200
TYPE AX5000_P_0200 :
STRUCT
	Actual_main_voltage_peak_value:UINT;
END_STRUCT
END_TYPE

// POUs/IO/Drives/SoE/Ax5000ParamSTRUCTs/P/AX5000_P_0201
TYPE AX5000_P_0201 :
STRUCT
	Nominal_main_voltage:UINT;
END_STRUCT
END_TYPE

// POUs/IO/Drives/SoE/Ax5000ParamSTRUCTs/P/AX5000_P_0202
TYPE AX5000_P_0202 :
STRUCT
	Main_voltage_positive_tolerance_range:UINT;
END_STRUCT
END_TYPE

// POUs/IO/Drives/SoE/Ax5000ParamSTRUCTs/P/AX5000_P_0203
TYPE AX5000_P_0203 :
STRUCT
	Main_voltage_negative_tolerance_range:UINT;
END_STRUCT
END_TYPE

// POUs/IO/Drives/SoE/Ax5000ParamSTRUCTs/P/AX5000_P_0204
TYPE AX5000_P_0204 :
STRUCT
	Power_management_control_word:UINT;
END_STRUCT
END_TYPE

// POUs/IO/Drives/SoE/Ax5000ParamSTRUCTs/P/AX5000_P_0205
TYPE AX5000_P_0205 :
STRUCT
	Power_management_status_word:UINT;
END_STRUCT
END_TYPE

// POUs/IO/Drives/SoE/Ax5000ParamSTRUCTs/P/AX5000_P_0206
{attribute 'pack_mode' := '1'}//Ensures 1-byte-alignmend
TYPE AX5000_P_0206 :
STRUCT
	Actual_lenght:UINT;
	Max_lenght:UINT;
	Umain_max_critical_hardware_voltage:UINT;
	Umain_min_critical_hardware_voltage:UINT;
	Umain_overvoltage_threshold:UINT;
	Umain_underervoltage_threshold:UINT;
	Umain_peak_overvoltage_threshold:UINT;
	Umain_peak_underervoltage_threshold:UINT;
	Umain_peak_lost_phase_threshold:UINT;
	Internal_brake_chopper_on_threshold:UINT;
	Internal_brake_chopper_off_threshold:UINT;
	Base_internal_brake_chopper_on_threshold:UINT;
	External_brake_chopper_on_threshold:UINT;
	External_brake_chopper_off_threshold:UINT;
	Base_external_brake_chopper_on_threshold:UINT;
	External_dc_link_connection_off_threshold:UINT;
	DCLink_volervoltage_on_threshold:UINT;
	DCLink_undervoltage_off_threshold:UINT;
	DCLink_undervoltage_warning_threshold:UINT;
	DCLink_undervoltage_error_threshold:UINT;
	DCLink_bypass_load_resistor_on_threshold:UINT;
	DCLink_bypass_load_resistor_off_threshold:UINT;
	External_Umain_rekay_off_threshold:UINT;
	External_Umain_rekay_on_threshold:UINT;
	AX5160_AX5193_Umain_peak_phase_monitoring_threshold:UINT;
//	{attribute 'hide'}
	Rsvd:ARRAY[0..6] OF UINT;

END_STRUCT
END_TYPE

// POUs/IO/Drives/SoE/Ax5000ParamSTRUCTs/P/AX5000_P_0207
{attribute 'pack_mode' := '1'}//Ensures 1-byte-alignmend
TYPE AX5000_P_0207 :
STRUCT
	Actual_lenght:UINT;
	Max_lenght:UINT;
	Resistance:UINT;
	Continuous_Power:UINT;
	Period_time_for_duty_cycle:UINT;
	Break_resistor_protection:UINT;
	Maximum_peak_energy_by_40Percent_duty_cycle:UDINT;
	Maximum_peak_energy_by_20Percent_duty_cycle:UDINT;
	Maximum_peak_energy_by_10Percent_duty_cycle:UDINT;
	Maximum_peak_energy_by_1Percent_duty_cycle:UDINT;
	Maximum_peak_energy_by_01Percent_duty_cycle:UDINT;
	Rsvd:ARRAY[0..3] OF UDINT;

END_STRUCT
END_TYPE

// POUs/IO/Drives/SoE/Ax5000ParamSTRUCTs/P/AX5000_P_0208
{attribute 'pack_mode' := '1'}//Ensures 1-byte-alignmend
TYPE AX5000_P_0208 :
STRUCT
	Actual_lenght:UINT;
	Max_lenght:UINT;
	Resistance:UINT;
	Continuous_Power:UINT;
	Period_time_for_duty_cycle:UINT;
	Break_resistor_protection:UINT;
	Maximum_peak_energy_by_40Percent_duty_cycle:UDINT;
	Maximum_peak_energy_by_20Percent_duty_cycle:UDINT;
	Maximum_peak_energy_by_10Percent_duty_cycle:UDINT;
	Maximum_peak_energy_by_1Percent_duty_cycle:UDINT;
	Maximum_peak_energy_by_01Percent_duty_cycle:UDINT;
	Rsvd:ARRAY[0..3] OF UDINT;

END_STRUCT
END_TYPE

// POUs/IO/Drives/SoE/Ax5000ParamSTRUCTs/P/AX5000_P_0209
TYPE AX5000_P_0209 :
STRUCT
	Internal_brak_resistor_actual_continouse_power:UINT;
END_STRUCT
END_TYPE

// POUs/IO/Drives/SoE/Ax5000ParamSTRUCTs/P/AX5000_P_0210
TYPE AX5000_P_0210 :
STRUCT
	External_brak_resistor_actual_continouse_power:UINT;
END_STRUCT
END_TYPE

// POUs/IO/Drives/SoE/Ax5000ParamSTRUCTs/P/AX5000_P_0211
TYPE AX5000_P_0211 :
STRUCT
	Warning_level_Actual_cont_power_internal_brake_resistor:UINT;
END_STRUCT
END_TYPE

// POUs/IO/Drives/SoE/Ax5000ParamSTRUCTs/P/AX5000_P_0212
TYPE AX5000_P_0212 :
STRUCT
	Warning_level_Actual_cont_power_external_brake_resistor:UINT;
END_STRUCT
END_TYPE

// POUs/IO/Drives/SoE/Ax5000ParamSTRUCTs/P/AX5000_P_0213
TYPE AX5000_P_0213 :
STRUCT
	External_DC_Link_current:DINT;
END_STRUCT
END_TYPE

// POUs/IO/Drives/SoE/Ax5000ParamSTRUCTs/P/AX5000_P_0214
TYPE AX5000_P_0214 :
STRUCT
	DC_Link_connection_mode:UINT;
END_STRUCT
END_TYPE

// POUs/IO/Drives/SoE/Ax5000ParamSTRUCTs/P/AX5000_P_0215
TYPE AX5000_P_0215 :
STRUCT
	Actual_Periphery_Voltage:UINT;
END_STRUCT
END_TYPE

// POUs/IO/Drives/SoE/Ax5000ParamSTRUCTs/P/AX5000_P_0216
TYPE AX5000_P_0216 :
STRUCT
	Max_DC_Link_voltage:UINT;
END_STRUCT
END_TYPE

// POUs/IO/Drives/SoE/Ax5000ParamSTRUCTs/P/AX5000_P_0217
TYPE AX5000_P_0217 :
STRUCT
	Actual_main_voltage:UINT;
END_STRUCT
END_TYPE

// POUs/IO/Drives/SoE/Ax5000ParamSTRUCTs/P/AX5000_P_0218
TYPE AX5000_P_0218 :
STRUCT
	Internal_brake_resistor_actual_peak_energy:UINT;
END_STRUCT
END_TYPE

// POUs/IO/Drives/SoE/Ax5000ParamSTRUCTs/P/AX5000_P_0219
TYPE AX5000_P_0219 :
STRUCT
	External_brake_resistor_actual_peak_energy:UINT;
END_STRUCT
END_TYPE

// POUs/IO/Drives/SoE/Ax5000ParamSTRUCTs/P/AX5000_P_0220
TYPE AX5000_P_0220 :
STRUCT
	Actual_lenght:UINT;
	Max_lenght:UINT;
	Max_energy_over_100percent_duty_cycle:UDINT;
	Max_energy_over_40percent_duty_cycle:UDINT;
	Max_energy_over_20percent_duty_cycle:UDINT;
	Max_energy_over_10percent_duty_cycle:UDINT;
	Max_energy_over_1percent_duty_cycle:UDINT;
	Max_energy_over_01percent_duty_cycle:UDINT;
END_STRUCT
END_TYPE

// POUs/IO/Drives/SoE/Ax5000ParamSTRUCTs/P/AX5000_P_0221
{attribute 'pack_mode' := '1'}//Ensures 1-byte-alignmend
TYPE AX5000_P_0221 :
STRUCT
	Actual_lenght:UINT;
	Max_lenght:UINT;
	Max_energy_over_100percent_duty_cycle:UDINT;
	Max_energy_over_40percent_duty_cycle:UDINT;
	Max_energy_over_20percent_duty_cycle:UDINT;
	Max_energy_over_10percent_duty_cycle:UDINT;
	Max_energy_over_1percent_duty_cycle:UDINT;
	Max_energy_over_01percent_duty_cycle:UDINT;
END_STRUCT
END_TYPE

// POUs/IO/Drives/SoE/Ax5000ParamSTRUCTs/P/AX5000_P_0250
TYPE AX5000_P_0250 :
STRUCT
	Scource:UINT;
END_STRUCT
END_TYPE

// POUs/IO/Drives/SoE/Ax5000ParamSTRUCTs/P/AX5000_P_0251
TYPE AX5000_P_0251 EXTENDS ST_AX5000_P_0251:
STRUCT
(*	Actual_lenght:UINT;
	Max_lenght:UINT;
	Mux1:UINT;
	Mux2:UINT;
	Logic:UINT;
	Latch_ctrl:UINT;
*)
END_STRUCT
END_TYPE

